// TIA Portal V19 export
FUNCTION_BLOCK "LAxisCtrlApcFr_Axis"   // FB19501, LAD
{ S7_Optimized_Access := 'TRUE' }
AUTHOR : APCFR
VERSION : 2.0
// V2.0.1
// stored: AutoNumber false, IsIECCheckEnabled true, MemoryReserve 100, SetENOAutomatically true
   VAR_INPUT
      enable : Bool := FALSE;
      stateSafetyActive : Bool := TRUE;   // STO or SOS active. Set FALSE if not used
      stateS120InfeedInOperation : Bool := FALSE;   // S120 infeed in operation input. Set TRUE if no infeed (AC/AC axis : CU310 or S210 or V90)
      enableAxis : Bool := FALSE;   // TRUE: Set axis enable; FALSE: Remove axis enable
      resetAxis : Bool := FALSE;   // Rising edge: Acknowledgement of technology alarms or restart of the axis (depending on configuration)
      openBrake : Bool := FALSE;
      jogForward : Bool := FALSE;   // Rising edge: Move an axis in jog mode (forward); Falling edge: Stop jogging
      jogBackward : Bool := FALSE;   // Rising edge: Move an axis in jog mode (backward); Falling edge: Stop jogging
      moveVelocity : Bool := FALSE;   // Rising edge: Move an axis at constant velocity/speed
      stop : Bool := FALSE;   // Rising edge: Brake an axis until it comes to a standstill
      eStop : Bool := FALSE;   // Emergency Stop with MC_Stop instruction
      torqueLimiting : Bool := FALSE;   // TRUE: Enable force/torque limiting
      homing : Bool := FALSE;   // Rising edge: Home axis
      homingToFixedStop : Bool := FALSE;
      homingOnSensor : Bool := FALSE;
      posRelative : Bool := FALSE;   // Rising edge: Move an axis relative to its position when execution of the job began
      posAbsolute : Bool := FALSE;   // Rising edge: Move an axis to an absolute position
      posSuperimposed : Bool := FALSE;   // Rising edge: Start a superimposed positioning
      haltSuperimposed : Bool := FALSE;
      gearInRelative : Bool := FALSE;
      gearInAbsolute : Bool := FALSE;
      gearInVelocity : Bool := FALSE;
      gearOutCamOut : Bool := FALSE;   // Rising edge: End a gearing/camming operation
      camIn : Bool := FALSE;
      camInStandStill : Bool := FALSE;
      camInChangeOnTheFly : Bool := FALSE;
      phasing : Bool := FALSE;
      offset : Bool := FALSE;   // Rising edge: Start an offset operation
      actDesactLimitSwitches : Bool := FALSE;
      changeModulo : Bool := FALSE;
      startEndLessMode : Bool := FALSE;
      simulationOnOff : Bool := FALSE;   // Rising edge starts action once
      resetMaxValues : Bool := FALSE;   // Reset max torque and max followingerror
      override : LReal := 100.0;   // Velocity override : 0 to 200%
      axis : DB_ANY;   // Reference to axis to be controlled
      master : DB_ANY;
      cam1 : DB_ANY;
      cam2 : DB_ANY;
      dataAxisConfig : "LAxisCtrlApcFr_typeAxisConfig";   // Structure for parameters
   END_VAR
   VAR_OUTPUT
      valid { ExternalWritable := 'False'} : Bool := FALSE;   // TRUE: Valid set of output values available at the FB
      busy { ExternalWritable := 'False'} : Bool := FALSE;
      error { ExternalWritable := 'False'} : Bool := FALSE;   // TRUE: An error occurred while processing the FB
      status { ExternalWritable := 'False'} : String := 'STATUS_NO_CALL';   // Current status of FB
      errorMC { ExternalWritable := 'False'} : String;
      errorID { ExternalWritable := 'False'} : String;
      driveReadyForOperation { ExternalWritable := 'False'} : Bool := FALSE;
      axisEnabled { ExternalWritable := 'False'} : Bool := FALSE;   // TRUE: The technology object is enabled. Motion commands can be executed
      axisHomed { ExternalWritable := 'False'} : Bool := FALSE;
      axisInPosition { ExternalWritable := 'False'} : Bool := FALSE;
      axisInStandstill { ExternalWritable := 'False'} : Bool := FALSE;
      axisInVelocity { ExternalWritable := 'False'} : Bool := FALSE;   // TRUE: The setpoint velocity/speed was reached and will be maintained
      axisInLimitation { ExternalWritable := 'False'} : Bool := FALSE;   // TRUE: The drive is operating at the force/torque limit
      axisInClamping { ExternalWritable := 'False'} : Bool := FALSE;   // TRUE: The drive is kept at the fixed stop (clamping), the axis position is within the positioning tolerance
      axisInSimulation : Bool := FALSE;
      axisCamInSelected { ExternalWritable := 'False'} : Bool := FALSE;
      axisInSynchronizing { ExternalWritable := 'False'} : Bool := FALSE;
      axisInSync { ExternalWritable := 'False'} : Bool := FALSE;
      camInStandStillDone { ExternalWritable := 'False'} : Bool := FALSE;
      camInStandStillBusy { ExternalWritable := 'False'} : Bool := FALSE;
      camInChangeOnTheFlyDone { ExternalWritable := 'False'} : Bool := FALSE;
      camInChangeOnTheFlylBusy { ExternalWritable := 'False'} : Bool := FALSE;
      eStopDone { ExternalWritable := 'False'} : Bool := FALSE;
      eStopBusy { ExternalWritable := 'False'} : Bool := FALSE;
      homingToFixedStopDone { ExternalWritable := 'False'} : Bool := FALSE;
      homingToFixedStopBusy { ExternalWritable := 'False'} : Bool := FALSE;
      homingOnSensorDone { ExternalWritable := 'False'} : Bool := FALSE;
      homingOnSensorBusy { ExternalWritable := 'False'} : Bool := FALSE;
      actDesactLimitSwitchesDone { ExternalWritable := 'False'} : Bool := FALSE;
      actDesactLimitSwitchesBusy { ExternalWritable := 'False'} : Bool := FALSE;
      changeModuloDone { ExternalWritable := 'False'} : Bool := FALSE;
      changeModuloBusy { ExternalWritable := 'False'} : Bool := FALSE;
      endLessModeDone { ExternalWritable := 'False'} : Bool := FALSE;
      endLessModeBusy { ExternalWritable := 'False'} : Bool := FALSE;
      simulationOnDone { ExternalWritable := 'False'} : Bool := FALSE;
      simulationOnBusy { ExternalWritable := 'False'} : Bool := FALSE;
      actualPosition { ExternalWritable := 'False'} : LReal;
      actualVelocity { ExternalWritable := 'False'} : LReal;
      actualSpeed { ExternalWritable := 'False'} : LReal;
      actualAcceleration { ExternalWritable := 'False'} : LReal;
      actualTorque { ExternalWritable := 'False'} : LReal;
      actualTorqueMax { ExternalWritable := 'False'} : LReal;
      actualFollowingError { ExternalWritable := 'False'} : LReal;
      actualFollowingErrorMax { ExternalWritable := 'False'} : LReal;
      camSelected { ExternalWritable := 'False'} : UInt;
      camUsed { ExternalWritable := 'False'} : UInt;
      HistoricBuffer { ExternalWritable := 'False'} : "LAxisCtrlApcFr_typeHistoricBufferCmd";
      outputsLAxisCtrl_Axis { ExternalWritable := 'False'} : Struct
         valid : Bool := FALSE;   // TRUE: Valid set of output values available at the FB
         busy : Bool := FALSE;   // TRUE: FB is working and new output values can be expected
         error : Bool := FALSE;   // TRUE: An error occurred while processing the FB
         status : Word;   // Current status of FB (16#0000 - 16#7FFF: Status of the FB, 16#8000 - 16#FFFF: Error identification)
         statusText : String := STRING#'STATUS_NO_CALL';   // Text of current status of FB
         subfunctionStatus : Word;   // Status of internally called subfunctions (ErrorID of Motion Control instructions)
         axisEnabled : Bool := FALSE;   // TRUE: The technology object is enabled. Motion commands can be executed
         resetActive : Bool := FALSE;   // TRUE: Reset/Restart of the axis is active
         commandBusy : Bool := FALSE;   // TRUE: The selected basic motion command is being executed
         commandDone : Bool := FALSE;   // TRUE: The selected basic motion command has completed without error
         commandAborted : Bool := FALSE;   // TRUE: The selected basic motion command has been aborted
         inVelocity : Bool := FALSE;   // TRUE: The setpoint velocity/speed was reached and will be maintained
         inLimitation : Bool := FALSE;   // TRUE: The drive is operating at the force/torque limit
         homingCommandBusy : Bool := FALSE;   // TRUE: Homing command is being executed
         homingCommandDone : Bool := FALSE;   // TRUE: Homing command has completed without error
         homingCommandAborted : Bool := FALSE;   // TRUE: Homing command has been aborted
         superimposedBusy : Bool := FALSE;   // TRUE: The selected superimposed motion command is being executed
         superimposedDone : Bool := FALSE;   // TRUE: The selected superimposed motion command has completed without error
         superimposedAborted : Bool := FALSE;   // TRUE: The selected superimposed motion command has been aborted
         superimposedStart : Bool := FALSE;   // TRUE: The selected superimposed motion is active
         inClamping : Bool := FALSE;   // TRUE: The drive is kept at the fixed stop (clamping), the axis position is within the positioning tolerance
         startSync : Bool := FALSE;   // TRUE: The axis is synchronizing to the leading axis / desynchronizing from the leading axis (Note: signal is only valid for the currently selected synchronous functionality, see outputs 'gearInRelativeSelected', 'gearInAbsoluteSelected', 'gearInVelocitySelected', 'gearOutCamOutSelected' or 'camInSelected')
         inSync : Bool := FALSE;   // TRUE: The axis is synchronized to the leading axis (Note: signal is only valid for the currently selected synchronous functionality, see outputs 'gearInRelativeSelected', 'gearInAbsoluteSelected', 'gearInVelocitySelected' or 'camInSelected')
         endOfProfile : Bool := FALSE;   // TRUE: The end of the cam has been reached. The output is displayed for at least one call when the cam is used cyclically
         inSimulation : Bool := FALSE;   // TRUE: Synchronous operation is being simulated
         jogSelected : Bool := FALSE;   // TRUE: Jogging is active
         moveVelocitySelected : Bool := FALSE;   // TRUE: Moving with constant velocity/speed is active
         stopSelected : Bool := FALSE;   // TRUE: Stopping is active
         fastStopSelected : Bool := FALSE;   // TRUE: Stopping is active (with fastStop dynamics)
         torqueLimitingSelected : Bool := FALSE;   // TRUE: Force/Torque limiting is active
         homingSelected : Bool := FALSE;   // TRUE: Homing is active
         posRelativeSelected : Bool := FALSE;   // TRUE: Relative positioning is active
         posAbsoluteSelected : Bool := FALSE;   // TRUE: Absolute positioning is active
         posSuperimposedSelected : Bool := FALSE;   // TRUE: Superimposed positioning is active (See also outputs: superimposedBusy, superimposedDone, superimposedAborted)
         haltSuperimposedSelected : Bool := FALSE;   // TRUE: Superimposed halting is active (See also outputs: superimposedBusy, superimposedDone, superimposedAborted)
         gearInRelativeSelected : Bool := FALSE;   // TRUE: Relative gearing is active (See also outputs: commandBusy, commandDone, commandAborted, inSync)
         gearInAbsoluteSelected : Bool := FALSE;   // TRUE: Absolute gearing is active (See also outputs: commandBusy, commandDone, commandAborted, startSync, inSync)
         gearInVelocitySelected : Bool := FALSE;   // TRUE: Velocity gearing is active (See also outputs: commandBusy, commandDone, commandAborted, startSync, inSync)
         gearOutCamOutSelected : Bool := FALSE;   // TRUE: End a gearing/camming operation is active (See also outputs: commandBusy, commandDone, commandAborted, startSync)
         camInSelected : Bool := FALSE;   // TRUE: Camming is active (See also outputs: commandBusy, commandDone, commandAborted, startSync, inSync)
         phasingSelected : Bool := FALSE;   // TRUE: Phasing is active (See also outputs: superimposedBusy, superimposedDone, superimposedAborted, superimposedStart)
         offsetSelected : Bool := FALSE;   // TRUE: Offset is active (See also outputs: superimposedBusy, superimposedDone, superimposedAborted, superimposedStart)
         diagnostics : "LAxisCtrl_typeDiagnostics";   // Diagnostics structure
      END_STRUCT;
      outputsStatusWordTO { ExternalWritable := 'False'} : Struct
         enable : Bool;   // TRUE: The technology object has been enabled
         error : Bool;   // TRUE: An error is present
         restartActive : Bool;   // TRUE: A restart is active. The technology object is being reinitialized
         onlineStartValuesChanged : Bool;   // TRUE: The restart tags have been changed. For the changes to be applied, the technology object must be reinitialized
         controlPanelActive : Bool;   // TRUE: The axis control panel is active
         homingDone : Bool;   // TRUE: The technology object is homed
         done : Bool;   // TRUE: No motion job is in progress and the axis control panel is deactivated
         standstill : Bool;   // TRUE: The axis is at a standstill
         positioningCommand : Bool;   // TRUE: A positioning command is active ("MC_MoveRelative", "MC_MoveAbsolute")
         jogCommand : Bool;   // TRUE: An "MC_MoveJog" job is running
         velocityCommand : Bool;   // TRUE: An "MC_MoveVelocity" job is running
         homingCommand : Bool;   // TRUE: An "MC_Home" job is being processed
         constantVelocity : Bool;   // TRUE: The velocity setpoint is reached. A constant velocity setpoint is output
         accelerating : Bool;   // TRUE: An acceleration operation is active
         decelerating : Bool;   // TRUE: A deceleration operation is active
         swLimitMinActive : Bool;   // TRUE: A negative software limit switch has been approached or exceeded
         swLimitMaxActive : Bool;   // TRUE: A positive software limit switch has been approached or exceeded
         hwLimitMinActive : Bool;   // TRUE: A negative hardware limit switch has been approached or exceeded
         hwLimitMaxActive : Bool;   // TRUE: A positive hardware limit switch has been approached or exceeded
         synchronizing : Bool;   // TRUE: The axis synchronizes to a leading value
         synchronous : Bool;   // TRUE: The axis moves synchronously to a leading value
         superimposedMotionCommand : Bool;   // TRUE: An "MC_MoveSuperimposed" job is running
         phasingCommand : Bool;   // TRUE: An "MC_PhasingAbsolute" or "MC_PhasingRelative" job for the leading value shift is active
         axisSimulation : Bool;   // TRUE: The technology object is in simulation
         torqueLimitingCommand : Bool;   // TRUE: An "MC_TorqueLimiting" job is running
         inLimitation : Bool;   // TRUE: The drive operates at least at the threshold value (default 90%) of the torque limit/force limitation
         nonPositionControlled : Bool;   // TRUE: The axis is not in position-controlled mode
         kinematicsMotionCommand : Bool;   // TRUE: The axis is used for a kinematics job
         inClamping : Bool;   // TRUE: The axis is clamped at a fixed stop
         motionInCommand : Bool;   // TRUE: An "MC_MotionIn" job is active
         stopCommand : Bool;   // TRUE: An "MC_Stop" job is running. The technology object is locked
         desynchronizingCommand : Bool;   // TRUE: An "MC_GearOut" job or "MC_CamOut" job is active. The following axis is desynchronized
         passingBacklash : Bool;   // TRUE: The backlash is traversed. <TO>.ActualPosition does not hereby change
         phasingCommandWaiting : Bool;   // TRUE: An "MC_PhasingAbsolute" or "MC_PhasingRelative" job for leading value shift is waiting
         offsetCommand : Bool;   // TRUE: An "MC_OffsetAbsolute" or "MC_OffsetRelative" job for following value offset is active
         offsetCommandWaiting : Bool;   // TRUE: An "MC_OffsetAbsolute" or "MC_OffsetRelative" job for following value offset is waiting
         motionInSuperimposedCommand : Bool;   // TRUE: An "MC_MotionInSuperimposed" job is running
         haltSuperimposedCommand : Bool;   // TRUE: An "MC_HaltSuperimposed" job is running
      END_STRUCT;
   END_VAR
   VAR
      statFirstCall { ExternalAccessible := 'False'; ExternalVisible := 'False'; ExternalWritable := 'False'} : Bool;   // TRUE: First call of FB
      statLastCall { ExternalAccessible := 'False'; ExternalVisible := 'False'; ExternalWritable := 'False'} : Bool;
      statEnableOld { ExternalAccessible := 'False'; ExternalVisible := 'False'; ExternalWritable := 'False'} : Bool;   // Old value of enable for edge detection
      statErrorLAxisCtrlStd { ExternalAccessible := 'False'; ExternalVisible := 'False'; ExternalWritable := 'False'} : Bool;
      statErrorActDesactLimitSwitches { ExternalAccessible := 'False'; ExternalVisible := 'False'; ExternalWritable := 'False'} : Bool;
      statErrorChangeModuloAxis { ExternalAccessible := 'False'; ExternalVisible := 'False'; ExternalWritable := 'False'} : Bool;
      statErrorHomingToFixedStop { ExternalAccessible := 'False'; ExternalVisible := 'False'; ExternalWritable := 'False'} : Bool;
      statErrorHomingOnSensor { ExternalAccessible := 'False'; ExternalVisible := 'False'; ExternalWritable := 'False'} : Bool;
      statErrorEndLessMode { ExternalAccessible := 'False'; ExternalVisible := 'False'; ExternalWritable := 'False'} : Bool;
      statErrorSimulationOnOff { ExternalAccessible := 'False'; ExternalVisible := 'False'; ExternalWritable := 'False'} : Bool;
      statErrorCamInStandStill { ExternalAccessible := 'False'; ExternalVisible := 'False'; ExternalWritable := 'False'} : Bool;
      statErrorCamSelection { ExternalAccessible := 'False'; ExternalVisible := 'False'; ExternalWritable := 'False'} : Bool;
      statErrorCamStandStillSelection { ExternalAccessible := 'False'; ExternalVisible := 'False'; ExternalWritable := 'False'} : Bool;
      statErrorInterpolateCam { ExternalAccessible := 'False'; ExternalVisible := 'False'; ExternalWritable := 'False'} : Bool;
      statErrorCamIChangeOnTheFly { ExternalAccessible := 'False'; ExternalVisible := 'False'; ExternalWritable := 'False'} : Bool;
      statErrorGearInPos { ExternalAccessible := 'False'; ExternalVisible := 'False'; ExternalWritable := 'False'} : Bool;
      statErrorEStop { ExternalAccessible := 'False'; ExternalVisible := 'False'; ExternalWritable := 'False'} : Bool;
      statFirstError { ExternalAccessible := 'False'; ExternalVisible := 'False'; ExternalWritable := 'False'} : Bool;
      returnValueRD_LOC_T { ExternalAccessible := 'False'; ExternalVisible := 'False'; ExternalWritable := 'False'} : Int;
      statEnableAxisOld { ExternalAccessible := 'False'; ExternalVisible := 'False'; ExternalWritable := 'False'} : Bool := FALSE;   // TRUE: Set axis enable; FALSE: Remove axis enable
      statHomingOld { ExternalAccessible := 'False'; ExternalVisible := 'False'; ExternalWritable := 'False'} : Bool := FALSE;   // Rising edge: Home axis
      statIndex { ExternalAccessible := 'False'; ExternalVisible := 'False'; ExternalWritable := 'False'} : Int;
      statHistoricBuffer { ExternalAccessible := 'False'; ExternalVisible := 'False'; ExternalWritable := 'False'} : "LAxisCtrlApcFr_typeHistoricBufferCmd";
      statAxisName { ExternalAccessible := 'False'; ExternalVisible := 'False'; ExternalWritable := 'False'} : WString;
      statDiagnostic { ExternalAccessible := 'False'; ExternalVisible := 'False'; ExternalWritable := 'False'} : Struct
         status : Word;
         errorMC : Word;
         errorID : Word;
      END_STRUCT;
      statReset { ExternalAccessible := 'False'; ExternalVisible := 'False'; ExternalWritable := 'False'} : Bool;
      statOpenBrake { ExternalAccessible := 'False'; ExternalVisible := 'False'; ExternalWritable := 'False'} : Bool;
      statStop { ExternalAccessible := 'False'; ExternalVisible := 'False'; ExternalWritable := 'False'} : Bool;
      statFastStop { ExternalAccessible := 'False'; ExternalVisible := 'False'; ExternalWritable := 'False'} : Bool;
      statEStop { ExternalAccessible := 'False'; ExternalVisible := 'False'; ExternalWritable := 'False'} : Bool;
      statTorqueLimiting { ExternalAccessible := 'False'; ExternalVisible := 'False'; ExternalWritable := 'False'} : Bool;
      statHoming { ExternalAccessible := 'False'; ExternalVisible := 'False'; ExternalWritable := 'False'} : Bool;
      statJogForward { ExternalAccessible := 'False'; ExternalVisible := 'False'; ExternalWritable := 'False'} : Bool;
      statJogBackward { ExternalAccessible := 'False'; ExternalVisible := 'False'; ExternalWritable := 'False'} : Bool;
      statMoveVelocity { ExternalAccessible := 'False'; ExternalVisible := 'False'; ExternalWritable := 'False'} : Bool;
      statPosRelative { ExternalAccessible := 'False'; ExternalVisible := 'False'; ExternalWritable := 'False'} : Bool;
      statPosAbsolute { ExternalAccessible := 'False'; ExternalVisible := 'False'; ExternalWritable := 'False'} : Bool;
      statSuperimposed { ExternalAccessible := 'False'; ExternalVisible := 'False'; ExternalWritable := 'False'} : Bool;
      statHaltSuperimposed { ExternalAccessible := 'False'; ExternalVisible := 'False'; ExternalWritable := 'False'} : Bool;
      statGearInVelocity { ExternalAccessible := 'False'; ExternalVisible := 'False'; ExternalWritable := 'False'} : Bool;
      statGearInRelative { ExternalAccessible := 'False'; ExternalVisible := 'False'; ExternalWritable := 'False'} : Bool;
      statGearInAbsolute { ExternalAccessible := 'False'; ExternalVisible := 'False'; ExternalWritable := 'False'} : Bool;
      statCamIn { ExternalAccessible := 'False'; ExternalVisible := 'False'; ExternalWritable := 'False'} : Bool;
      statCamInStandStill { ExternalAccessible := 'False'; ExternalVisible := 'False'; ExternalWritable := 'False'} : Bool;
      statCamInChangeOnTheFly { ExternalAccessible := 'False'; ExternalVisible := 'False'; ExternalWritable := 'False'} : Bool;
      statGearOutCamOut { ExternalAccessible := 'False'; ExternalVisible := 'False'; ExternalWritable := 'False'} : Bool;
      statPhasing { ExternalAccessible := 'False'; ExternalVisible := 'False'; ExternalWritable := 'False'} : Bool;
      statOffset { ExternalAccessible := 'False'; ExternalVisible := 'False'; ExternalWritable := 'False'} : Bool;
      statCam { ExternalAccessible := 'False'; ExternalVisible := 'False'; ExternalWritable := 'False'} : DB_ANY;
      statCamStandStill { ExternalAccessible := 'False'; ExternalVisible := 'False'; ExternalWritable := 'False'} : DB_ANY;
      statCamStanStillSelected { ExternalAccessible := 'False'; ExternalVisible := 'False'; ExternalWritable := 'False'} : UInt;
      statActDesactLimitSwitches { ExternalAccessible := 'False'; ExternalVisible := 'False'; ExternalWritable := 'False'} : Bool;
      statChangeModulo { ExternalAccessible := 'False'; ExternalVisible := 'False'; ExternalWritable := 'False'} : Bool;
      statHomingToFixedStop { ExternalAccessible := 'False'; ExternalVisible := 'False'; ExternalWritable := 'False'} : Bool;
      statHomingOnSensor { ExternalAccessible := 'False'; ExternalVisible := 'False'; ExternalWritable := 'False'} : Bool;
      statStartEndLessMode { ExternalAccessible := 'False'; ExternalVisible := 'False'; ExternalWritable := 'False'} : Bool;
      statSimulationOnOff { ExternalAccessible := 'False'; ExternalVisible := 'False'; ExternalWritable := 'False'} : Bool;
      statDataAxisConfigLAxisCtrl { ExternalAccessible := 'False'; ExternalVisible := 'False'; ExternalWritable := 'False'} : "LAxisCtrl_typeAxisConfig";
      statOffsetChangeOnTheFly { ExternalAccessible := 'False'; ExternalVisible := 'False'; ExternalWritable := 'False'} : LReal;
      statAxisCommandStatusDWord : DWord;
      instLAxisCtrl_Axis { ExternalAccessible := 'False'; ExternalVisible := 'False'; ExternalWritable := 'False'} : "LAxisCtrl_Axis";
      instLAxisCtrl_AxisStatusWord { ExternalAccessible := 'False'; ExternalVisible := 'False'; ExternalWritable := 'False'} : "LAxisCtrl_AxisStatusWord";
      instLAxisCtrlApcFr_CamInStandStill { ExternalAccessible := 'False'; ExternalVisible := 'False'; ExternalWritable := 'False'} : "LAxisCtrlApcFr_CamInStandStill";
      instLAxisCtrlApcFr_GetCamStatusWord { ExternalAccessible := 'False'; ExternalVisible := 'False'; ExternalWritable := 'False'} : "LAxisCtrlApcFr_UnpubGetCamStatusWord";
      InstLAxisCtrlApcFr_McGearInPos_Axis { ExternalAccessible := 'False'; ExternalVisible := 'False'; ExternalWritable := 'False'} : "LAxisCtrlApcFr_McGearInPos_Axis";
      instLAxisCtrlApcFr_HystoricBuffer { ExternalAccessible := 'False'; ExternalVisible := 'False'; ExternalWritable := 'False'} : "LAxisCtrlApcFr_HystoricBuffer";
      instLAxisCtrlApcFr_UnpubAxis_eSTOP { ExternalAccessible := 'False'; ExternalVisible := 'False'; ExternalWritable := 'False'} : "LAxisCtrlApcFr_UnpubAxis_eSTOP";
      instLaxisCtrlApcFr_GetCommandAxisStatusDWord { ExternalAccessible := 'False'; ExternalVisible := 'False'; ExternalWritable := 'False'} : "LAxisCtrlApcFr_GetCommandAxisStatusDWord";
      instLaxisCtrlApcFr_UnpubMC_Interpolate { ExternalAccessible := 'False'; ExternalVisible := 'False'; ExternalWritable := 'False'} : "LAxisCtrlApcFr_UnpubMC_Interpolate";
      instLAxisCtrlApcFr_ActDeactLimitSwitches { ExternalAccessible := 'False'; ExternalVisible := 'False'; ExternalWritable := 'False'} : "LAxisCtrlApcFr_ActDeactLimitSwitches";
      instLAxisCtrlApcFr_ChangeModulo { ExternalAccessible := 'False'; ExternalVisible := 'False'; ExternalWritable := 'False'} : "LAxisCtrlApcFr_ChangeModulo";
      instLAxisCtrlApcFr_HomingToFixedStop { ExternalAccessible := 'False'; ExternalVisible := 'False'; ExternalWritable := 'False'} : "LAxisCtrlApcFr_HomingToFixedStop";
      instAxisCtrlAapcFr_HomingOnSensor { ExternalAccessible := 'False'; ExternalVisible := 'False'; ExternalWritable := 'False'} : "LAxisCtrlApcFr_HomingOnSensor";
      instLAxisCtrlApcFr_EndLessMode { ExternalAccessible := 'False'; ExternalVisible := 'False'; ExternalWritable := 'False'} : "LAxisCtrlApcFr_EndLessMode";
      instLAxisCtrlApcFR_SimulationOnOff { ExternalAccessible := 'False'; ExternalVisible := 'False'; ExternalWritable := 'False'} : "LAxisCtrlApcFr_SimulationOnOff";
      instLaxisCtrlApcFr_CamInChangeOnTheFly { ExternalAccessible := 'False'; ExternalVisible := 'False'; ExternalWritable := 'False'} : "LAxisCtrlApcFr_CamInChangeOnTheFly";
      statAxis { ExternalAccessible := 'False'; ExternalVisible := 'False'; ExternalWritable := 'False'} : DB_ANY;
      statMaster { ExternalAccessible := 'False'; ExternalVisible := 'False'; ExternalWritable := 'False'} : DB_ANY;
      statCommunicationOK { ExternalAccessible := 'False'; ExternalVisible := 'False'; ExternalWritable := 'False'} : Bool;
   END_VAR
   VAR_TEMP
      tempVoidBool : Bool;   // Temp value for operative sensor
      tempAbsActualTorque : LReal;
      tempAbsActualTorqueMax : LReal;
      tempRefCamBase2 : REF_TO TO_CamBase;   // Temporary reference of the technology object type TO_CamBase
      tempRefCamBase1 : REF_TO TO_CamBase;   // Temporary reference of the technology object type TO_CamBase
      tempRefAxis : REF_TO TO_Axis;   // Temporary reference of the technology object type TO_Axis
      tempRefSpeedAxis : REF_TO TO_SpeedAxis;   // Temporary reference of the technology object type TO_SpeedAxis
      tempRefPosAxis : REF_TO TO_PositioningAxis;   // Temporary reference of the technology object type TO_PositioningAxis
      tempRefSyncAxis : REF_TO TO_SynchronousAxis;   // Temporary reference of the technology object type TO_PositioningAxis
      tempReturnValue : Int;
      tempDateAndTime : Date_And_Time;
      tempDateOfDay : Time_Of_Day;
   END_VAR
   VAR_TEMP   // added for the SCL form of the ladder/FBD networks
      _w1 : Bool;
   END_VAR
BEGIN

REGION Network 1 (SCL): (** COMMENTS **)
   //===================================================================================================
   // SIEMENS SAS    RC-FR DI FA APC
   //---------------------------------------------------------------------------------------------------
   // Restrictions:  TIA V16 or more in function of library version
   // Requirements:  S7-1500 + LAxisCtrl library
   //---------------------------------------------------------------------------------------------------
   // Description:   This function block offers basic functionalities for TO SynchronousAxis
   //                based on LAxisCtrl_SyncAxisCamming with additionnals functionalities
   //---------------------------------------------------------------------------------------------------
   // Change log table:
   // Version  Date        TIA   Expert  Changes applied
   // 01.xx    2020.07.24  V16   SDA     see LaxisCtrlApcFr_aVersion 
   // 02.xx    2021.10.18  V17   SDA     see LaxisCtrlApcFr_aVersion 
   // 03.xx    2024.09.12  V19   SDA     see LaxisCtrlApcFr_aVersion
   //---------------------------------------------------------------------------------------------------
   // Compatibility to TIA version require the use of latest version for PLC fimware and Motion Control 
   // e.g: Firmware 3.1 and Motion Control V7.0 for TIA V19
   //===================================================================================================
END_REGION

REGION Network 2 (SCL): (** INIT **)
   //----------------------------------------------------------------------------------------------
   #statFirstCall := #enable AND NOT #statEnableOld;
   #statLastCall := NOT #enable AND #statEnableOld;
   #statEnableOld := #enable;

   #tempRefAxis ?= #master;
   #tempRefSyncAxis ?= #axis;
   #tempRefCamBase1 ?= #cam1;
   #tempRefCamBase2 ?= #cam2;

   #statAxis := #axis;
   #statMaster := #master;

   IF #statFirstCall THEN
       REGION InitFirstCall
           // #statAxisName := GetSymbolPath(variable := #axis, size := 36);
           // "LaxisCtrlApcFr_GetPosSyncAxisGeneralValues"(axis := #axis,
           // axisGeneral := #dataAxisConfig.axisGeneral);
           // Diagnostic in string
           #status := 'STATUS_FIRST_CALL';
           #error := FALSE;
           #errorMC := 'No errorMC';
           #errorID := 'No errorID';
           // Diagnostic in word
           #statDiagnostic.status := "STATUS_FIRST_CALL";
           #statDiagnostic.errorMC := "STATUS_FINISHED_NOERROR";
           #statDiagnostic.errorID := "STATUS_FINISHED_NOERROR";

           #statFirstError := FALSE;

           #statAxis := #axis;
           #statMaster := #master;
           RETURN;
       END_REGION

   ELSIF #statLastCall THEN
       REGION InitLastCall
           // Reset outputs
           REGION Reset outputs 
               #error := FALSE;
               #status := 'STATUS_LAST_CALL';
               #errorMC := 'No ErrorMC';
               #statDiagnostic.status := "STATUS_FINISHED_NOERROR";
               #statDiagnostic.errorMC := "STATUS_FINISHED_NOERROR";
               #driveReadyForOperation := FALSE;
               #axisInPosition := FALSE;
               #axisInStandstill := FALSE;
               #axisInVelocity := FALSE;
               #axisInLimitation := FALSE;
               #axisInClamping := FALSE;
               #axisCamInSelected := FALSE;
               #axisInSynchronizing := FALSE;
               #camInStandStillDone := FALSE;
               #camInStandStillBusy := FALSE;
               #camInChangeOnTheFlyDone := FALSE;
               #camInChangeOnTheFlylBusy := FALSE;
               #axisInSync := FALSE;
               #eStopDone := FALSE;
               #eStopBusy := FALSE;
               #homingToFixedStopDone := FALSE;
               #homingToFixedStopBusy := FALSE;
               #homingOnSensorDone := FALSE;
               #homingOnSensorBusy := FALSE;
               #actDesactLimitSwitchesDone := FALSE;
               #actDesactLimitSwitchesBusy := FALSE;
               #changeModuloDone := FALSE;
               #changeModuloBusy := FALSE;
               #endLessModeDone := FALSE;
               #endLessModeBusy := FALSE;
               #simulationOnDone := FALSE;
               #simulationOnBusy := FALSE;
               #actualPosition := 0.0;
               #actualVelocity := 0.0;
               #actualSpeed := 0.0;
               #actualAcceleration := 0.0;
               #actualTorque := 0.0;
               #actualTorqueMax := 0.0;
               #actualFollowingError := 0.0;
               #actualFollowingErrorMax := 0.0;
           END_REGION

           // Reset internal variables
           REGION Reset internal variables
               #statFirstCall := FALSE;
               #statLastCall := FALSE;
               #statEnableOld := FALSE;
               #statErrorLAxisCtrlStd := FALSE;
               #statErrorActDesactLimitSwitches := FALSE;
               #statErrorChangeModuloAxis := FALSE;
               #statErrorHomingToFixedStop := FALSE;
               #statErrorHomingOnSensor := FALSE;
               #statErrorEndLessMode := FALSE;
               #statErrorEStop := FALSE;
               #statFirstError := FALSE;
               #statEnableAxisOld := FALSE;
               #statHomingOld := FALSE;
               #statIndex := 0;
               #statReset := FALSE;
               #statOpenBrake := FALSE;
               #statStop := FALSE;
               #statFastStop := FALSE;
               #statEStop := FALSE;
               #statTorqueLimiting := FALSE;
               #statHoming := FALSE;
               #statJogForward := FALSE;
               #statJogBackward := FALSE;
               #statMoveVelocity := FALSE;
               #statPosRelative := FALSE;
               #statPosAbsolute := FALSE;
               #statSuperimposed := FALSE;
               #statHaltSuperimposed := FALSE;
               #statGearInRelative := FALSE;
               // cpu-t functions
               #statGearInVelocity := FALSE;
               #statGearInAbsolute := FALSE;
               #statGearInAbsolute := FALSE;
               #statCamInStandStill := FALSE;
               #statCamInChangeOnTheFly := FALSE;
               #statGearOutCamOut := FALSE;
               #statPhasing := FALSE;
               #statOffset := FALSE;
               // additionnal functions
               #statActDesactLimitSwitches := FALSE;
               #statChangeModulo := FALSE;
               #statHomingToFixedStop := FALSE;
               #statHomingOnSensor := FALSE;
               #statStartEndLessMode := FALSE;
               #statSimulationOnOff := FALSE;
           END_REGION

           //RETURN;
       END_REGION

   ELSIF NOT #enable AND NOT #instLAxisCtrl_Axis.busy THEN
       REGION NotEnable

           #error := FALSE;
           // Diagnostic in string
           #status := 'STATUS_NO_CALL';
           #errorMC := 'No errorMC';
           #errorID := 'No errorID';
           // Diagnostic in word
           #statDiagnostic.status := "STATUS_NO_CALL";
           #statDiagnostic.errorMC := "STATUS_FINISHED_NOERROR";
           #statDiagnostic.errorID := "STATUS_FINISHED_NOERROR";
           #statFirstError := FALSE;

           RETURN;
       END_REGION
   END_IF;

   IF NOT #error THEN
       #status := 'STATUS_CALL_FB';
       #errorMC := 'No errorMC';
       #statDiagnostic.status := "STATUS_FINISHED_NOERROR";
       #statDiagnostic.errorMC := "STATUS_FINISHED_NOERROR";
   END_IF;
   //----------------------------------------------------------------------------------------------
END_REGION

REGION Network 3 (SCL): (** COMMAND **)
   IF #enable AND NOT #error THEN
       #statReset := #resetAxis;
       #statOpenBrake := #openBrake;
       #statStop := #stop;
       //#statFastStop := #fastStop;
       #statTorqueLimiting := #torqueLimiting;
       #statHoming := #homing;
       #statJogForward := #jogForward;
       #statJogBackward := #jogBackward;
       #statMoveVelocity := #moveVelocity;
       #statPosRelative := #posRelative;
       #statPosAbsolute := #posAbsolute;
       #statSuperimposed := #posSuperimposed;
       #statHaltSuperimposed := #haltSuperimposed;
       #statGearInRelative := #gearInRelative;
       #statCamIn := #camIn;
       #statGearOutCamOut := #gearOutCamOut;
       #statPhasing := #phasing;
       #statOffset := #offset;

       #statGearInAbsolute := #gearInAbsolute;
       #statGearInVelocity := #gearInVelocity;
       #statCamInStandStill := #camInStandStill;
       #statCamInChangeOnTheFly := #camInChangeOnTheFly;
       #statEStop := #eStop;
       #statActDesactLimitSwitches := #actDesactLimitSwitches;
       #statChangeModulo := #changeModulo;
       #statHomingToFixedStop := #homingToFixedStop;
       #statHomingOnSensor := #homingOnSensor;
       #statStartEndLessMode := #startEndLessMode;
       #statSimulationOnOff := #simulationOnOff;

   ELSIF #error THEN
       #statReset := #resetAxis;
       #statOpenBrake := #openBrake;
       #statStop := #stop;
       //#statFastStop := #fastStop;
       #statTorqueLimiting := FALSE;
       #statHoming := FALSE;
       #statJogForward := FALSE;
       #statJogBackward := FALSE;
       #statMoveVelocity := FALSE;
       #statPosRelative := FALSE;
       #statPosAbsolute := FALSE;
       #statSuperimposed := FALSE;
       #statHaltSuperimposed := FALSE;

       #statGearInRelative := FALSE;
       #statCamIn := FALSE;
       #statGearOutCamOut := FALSE;
       #statPhasing := FALSE;
       #statOffset := FALSE;

       #statGearInAbsolute := FALSE;
       #statGearInVelocity := FALSE;
       #statCamInStandStill := FALSE;
       #statCamInChangeOnTheFly := FALSE;
       #statEStop := #eStop;
       #statActDesactLimitSwitches := FALSE;
       #statChangeModulo := FALSE;
       #statHomingToFixedStop := FALSE;
       #statHomingOnSensor := FALSE;
       #statStartEndLessMode := FALSE;
       #statSimulationOnOff := FALSE;

    ELSE
        #statReset := FALSE;
        #statOpenBrake := FALSE;
        #statStop := FALSE;
        #statFastStop := FALSE;
        #statEStop := false;
        #statTorqueLimiting := FALSE;
        #statHoming := FALSE;
        #statJogForward := FALSE;
        #statJogBackward := FALSE;
        #statMoveVelocity := FALSE;
        #statPosRelative := FALSE;
        #statPosAbsolute := FALSE;
        #statSuperimposed := FALSE;
        #statHaltSuperimposed := FALSE;

        #statGearInRelative := FALSE;
        #statCamIn := FALSE;
        #statGearOutCamOut := FALSE;
        #statPhasing := FALSE;
        #statOffset := FALSE;

        #statGearInAbsolute := FALSE;
        #statGearInVelocity := FALSE;
        #statCamInStandStill := FALSE;
        #statCamInChangeOnTheFly := FALSE;
        #statEStop := FALSE;
        #statActDesactLimitSwitches := FALSE;
        #statChangeModulo := FALSE;
        #statHomingToFixedStop := FALSE;
        #statHomingOnSensor := FALSE;
        #statStartEndLessMode := FALSE;
        #statSimulationOnOff := FALSE;

   END_IF;
END_REGION

REGION Network 4: (** INTERPOLATE CAM **) / (** HISTORIC BUFFER **)
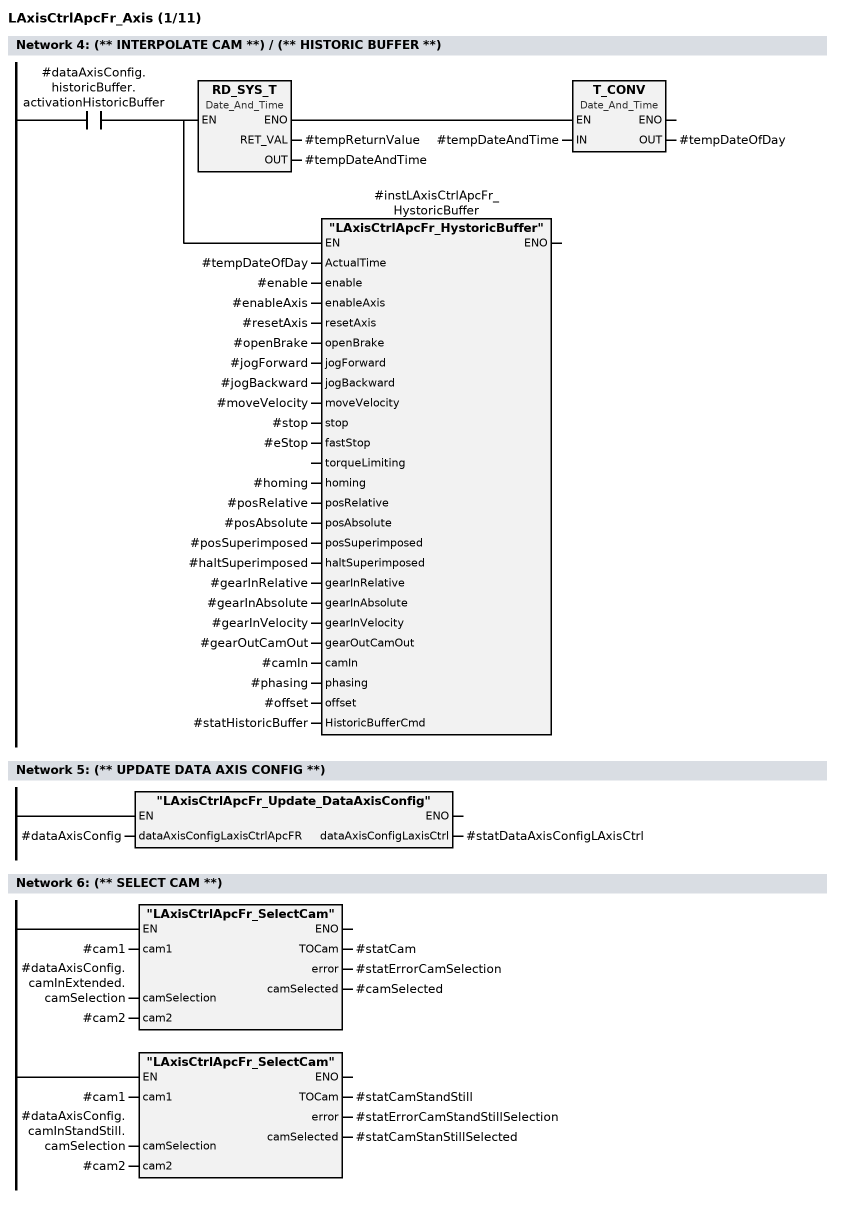
   RUNG wire#powerrail
      Contact( #dataAxisConfig.historicBuffer.activationHistoricBuffer )
      wire#w1
      { S7_Templates := "date_type := Date_And_Time" } RD_SYS_T(RET_VAL => #tempReturnValue, OUT => #tempDateAndTime)
      { S7_Templates := "[src_type := Date_And_Time, dest_type := Time_Of_Day]" } T_CONV(IN := #tempDateAndTime, OUT => #tempDateOfDay)
   END_RUNG
   RUNG wire#w1
      #instLAxisCtrlApcFr_HystoricBuffer(ActualTime := #tempDateOfDay, enable := #enable, enableAxis := #enableAxis, resetAxis := #resetAxis, openBrake := #openBrake, jogForward := #jogForward, jogBackward := #jogBackward, moveVelocity := #moveVelocity, stop := #stop, fastStop := #eStop, torqueLimiting :=, homing := #homing, posRelative := #posRelative, posAbsolute := #posAbsolute, posSuperimposed := #posSuperimposed, haltSuperimposed := #haltSuperimposed, gearInRelative := #gearInRelative, gearInAbsolute := #gearInAbsolute, gearInVelocity := #gearInVelocity, gearOutCamOut := #gearOutCamOut, camIn := #camIn, phasing := #phasing, offset := #offset, HistoricBufferCmd := #statHistoricBuffer)
   END_RUNG
   // the same network as SCL:
   #tempReturnValue := RD_SYS_T(EN := #dataAxisConfig.historicBuffer.activationHistoricBuffer,
                           OUT => #tempDateAndTime,
                           ENO => #_w1);
   IF #_w1 THEN T_CONV(IN := #tempDateAndTime, OUT => #tempDateOfDay); END_IF;
   IF #dataAxisConfig.historicBuffer.activationHistoricBuffer THEN
       #instLAxisCtrlApcFr_HystoricBuffer(ActualTime := #tempDateOfDay,   // "LAxisCtrlApcFr_HystoricBuffer"
                               enable := #enable,
                               enableAxis := #enableAxis,
                               resetAxis := #resetAxis,
                               openBrake := #openBrake,
                               jogForward := #jogForward,
                               jogBackward := #jogBackward,
                               moveVelocity := #moveVelocity,
                               stop := #stop,
                               fastStop := #eStop,
                               homing := #homing,
                               posRelative := #posRelative,
                               posAbsolute := #posAbsolute,
                               posSuperimposed := #posSuperimposed,
                               haltSuperimposed := #haltSuperimposed,
                               gearInRelative := #gearInRelative,
                               gearInAbsolute := #gearInAbsolute,
                               gearInVelocity := #gearInVelocity,
                               gearOutCamOut := #gearOutCamOut,
                               camIn := #camIn,
                               phasing := #phasing,
                               offset := #offset,
                               HistoricBufferCmd := #statHistoricBuffer);
   END_IF;
END_REGION

REGION Network 5: (** UPDATE DATA AXIS CONFIG **)
   RUNG wire#powerrail
      "LAxisCtrlApcFr_Update_DataAxisConfig"(dataAxisConfigLaxisCtrlApcFR := #dataAxisConfig, dataAxisConfigLaxisCtrl => #statDataAxisConfigLAxisCtrl)
   END_RUNG
   // the same network as SCL:
   "LAxisCtrlApcFr_Update_DataAxisConfig"(dataAxisConfigLaxisCtrlApcFR := #dataAxisConfig,
                           dataAxisConfigLaxisCtrl => #statDataAxisConfigLAxisCtrl);
END_REGION

REGION Network 6: (** SELECT CAM **)
   RUNG wire#powerrail
      "LAxisCtrlApcFr_SelectCam"(cam1 := #cam1, camSelection := #dataAxisConfig.camInExtended.camSelection, cam2 := #cam2, TOCam => #statCam, error => #statErrorCamSelection, camSelected => #camSelected)
   END_RUNG
   RUNG wire#powerrail
      "LAxisCtrlApcFr_SelectCam"(cam1 := #cam1, camSelection := #dataAxisConfig.camInStandStill.camSelection, cam2 := #cam2, TOCam => #statCamStandStill, error => #statErrorCamStandStillSelection, camSelected => #statCamStanStillSelected)
   END_RUNG
   // the same network as SCL:
   "LAxisCtrlApcFr_SelectCam"(cam1 := #cam1,
                           camSelection := #dataAxisConfig.camInExtended.camSelection,
                           cam2 := #cam2,
                           TOCam => #statCam,
                           error => #statErrorCamSelection,
                           camSelected => #camSelected);
   "LAxisCtrlApcFr_SelectCam"(cam1 := #cam1,
                           camSelection := #dataAxisConfig.camInStandStill.camSelection,
                           cam2 := #cam2,
                           TOCam => #statCamStandStill,
                           error => #statErrorCamStandStillSelection,
                           camSelected => #statCamStanStillSelected);
END_REGION

REGION Network 7: (** INTERPOLATE CAM **)
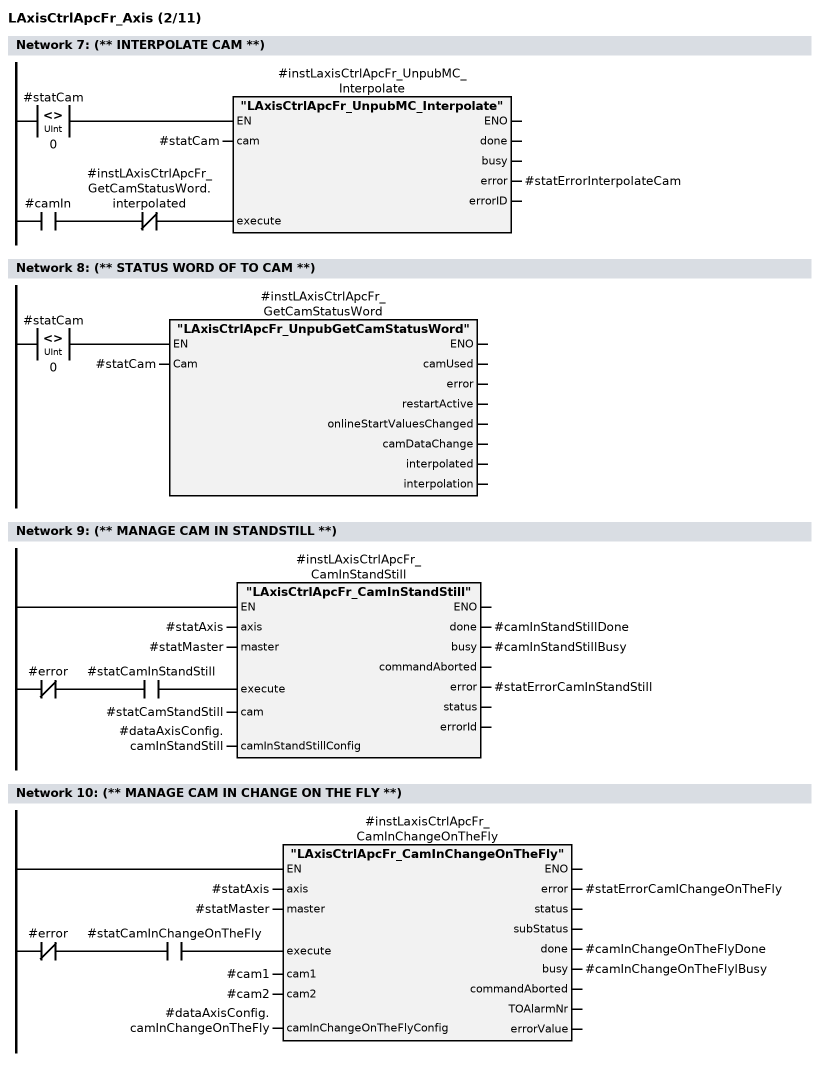
   RUNG wire#powerrail
      { S7_Templates := "SrcType := UInt" } NE_Contact(in1 := #statCam, in2 := 0)
      #instLaxisCtrlApcFr_UnpubMC_Interpolate(execute := wire#w1, cam := #statCam, done =>, busy =>, error => #statErrorInterpolateCam, errorID =>)
   END_RUNG
   RUNG wire#powerrail
      Contact( #camIn )
      I_Contact( #instLAxisCtrlApcFr_GetCamStatusWord.interpolated )
   END_RUNG wire#w1
   // the same network as SCL:
   IF #statCam <> 0 THEN
       #instLaxisCtrlApcFr_UnpubMC_Interpolate(cam := #statCam,   // "LAxisCtrlApcFr_UnpubMC_Interpolate"
                               execute := #camIn AND NOT #instLAxisCtrlApcFr_GetCamStatusWord.interpolated,
                               error => #statErrorInterpolateCam);
   END_IF;
END_REGION

REGION Network 8: (** STATUS WORD OF TO CAM **)
   RUNG wire#powerrail
      { S7_Templates := "SrcType := UInt" } NE_Contact(in1 := #statCam, in2 := 0)
      #instLAxisCtrlApcFr_GetCamStatusWord(Cam := #statCam, camUsed =>, error =>, restartActive =>, onlineStartValuesChanged =>, camDataChange =>, interpolated =>, interpolation =>)
   END_RUNG
   // the same network as SCL:
   IF #statCam <> 0 THEN
       #instLAxisCtrlApcFr_GetCamStatusWord(Cam := #statCam);   // "LAxisCtrlApcFr_UnpubGetCamStatusWord"
   END_IF;
END_REGION

REGION Network 9: (** MANAGE CAM IN STANDSTILL **)
   RUNG wire#powerrail
      #instLAxisCtrlApcFr_CamInStandStill(execute := wire#w1, axis := #statAxis, master := #statMaster, cam := #statCamStandStill, camInStandStillConfig := #dataAxisConfig.camInStandStill, done => #camInStandStillDone, busy => #camInStandStillBusy, commandAborted =>, error => #statErrorCamInStandStill, status =>, errorId =>)
   END_RUNG
   RUNG wire#powerrail
      I_Contact( #error )
      Contact( #statCamInStandStill )
   END_RUNG wire#w1
   // the same network as SCL:
   #instLAxisCtrlApcFr_CamInStandStill(axis := #statAxis,   // "LAxisCtrlApcFr_CamInStandStill"
                           master := #statMaster,
                           execute := NOT #error AND #statCamInStandStill,
                           cam := #statCamStandStill,
                           camInStandStillConfig := #dataAxisConfig.camInStandStill,
                           done => #camInStandStillDone,
                           busy => #camInStandStillBusy,
                           error => #statErrorCamInStandStill);
END_REGION

REGION Network 10: (** MANAGE CAM IN CHANGE ON THE FLY **)
   RUNG wire#powerrail
      #instLaxisCtrlApcFr_CamInChangeOnTheFly(execute := wire#w1, axis := #statAxis, master := #statMaster, cam1 := #cam1, cam2 := #cam2, camInChangeOnTheFlyConfig := #dataAxisConfig.camInChangeOnTheFly, error => #statErrorCamIChangeOnTheFly, status =>, subStatus =>, done => #camInChangeOnTheFlyDone, busy => #camInChangeOnTheFlylBusy, commandAborted =>, TOAlarmNr =>, errorValue =>)
   END_RUNG
   RUNG wire#powerrail
      I_Contact( #error )
      Contact( #statCamInChangeOnTheFly )
   END_RUNG wire#w1
   // the same network as SCL:
   #instLaxisCtrlApcFr_CamInChangeOnTheFly(axis := #statAxis,   // "LAxisCtrlApcFr_CamInChangeOnTheFly"
                           master := #statMaster,
                           execute := NOT #error AND #statCamInChangeOnTheFly,
                           cam1 := #cam1,
                           cam2 := #cam2,
                           camInChangeOnTheFlyConfig := #dataAxisConfig.camInChangeOnTheFly,
                           error => #statErrorCamIChangeOnTheFly,
                           done => #camInChangeOnTheFlyDone,
                           busy => #camInChangeOnTheFlylBusy);
END_REGION

REGION Network 11: (** CALL LAXISCTRL STD SYNC CAMMING **) / (** CALL LAXISCTRL AXIS **)
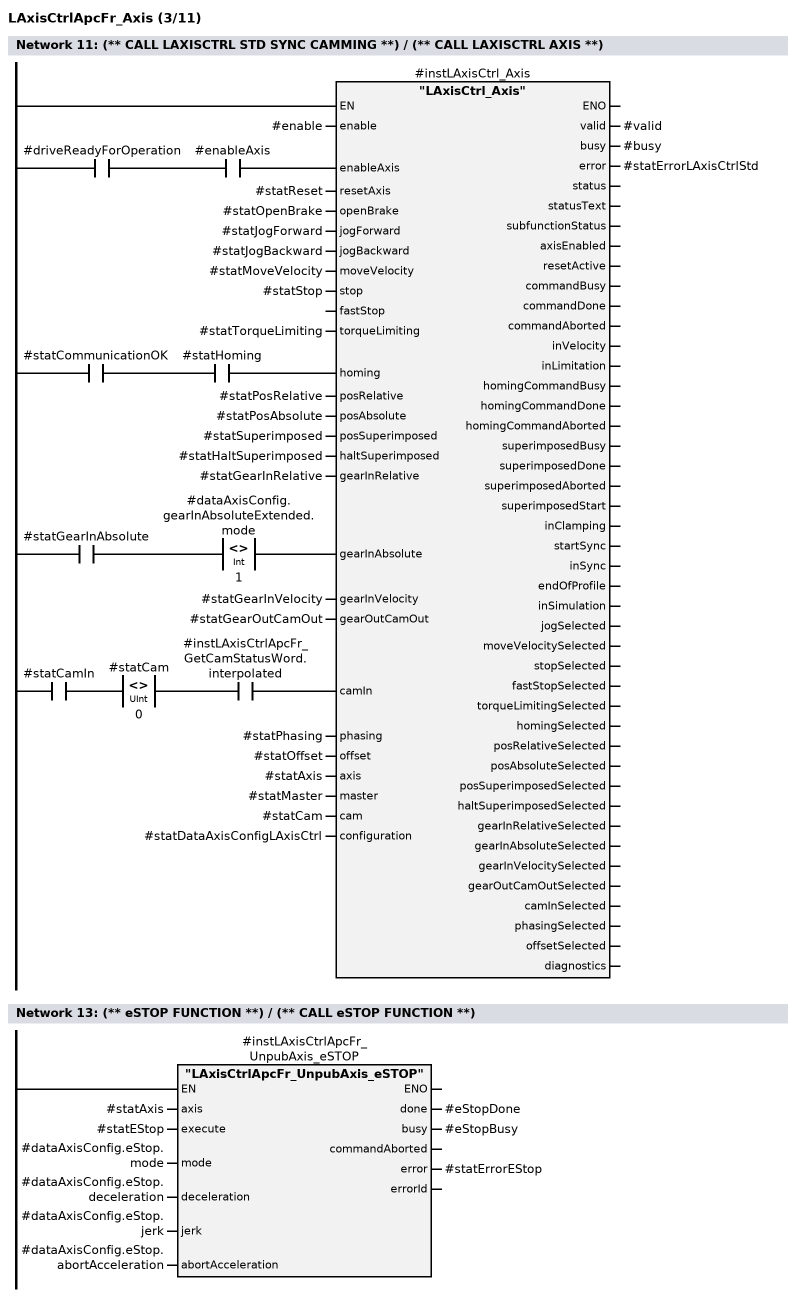
   RUNG wire#powerrail
      #instLAxisCtrl_Axis(enableAxis := wire#w1, homing := wire#w2, gearInAbsolute := wire#w3, camIn := wire#w4, enable := #enable, resetAxis := #statReset, openBrake := #statOpenBrake, jogForward := #statJogForward, jogBackward := #statJogBackward, moveVelocity := #statMoveVelocity, stop := #statStop, fastStop :=, torqueLimiting := #statTorqueLimiting, posRelative := #statPosRelative, posAbsolute := #statPosAbsolute, posSuperimposed := #statSuperimposed, haltSuperimposed := #statHaltSuperimposed, gearInRelative := #statGearInRelative, gearInVelocity := #statGearInVelocity, gearOutCamOut := #statGearOutCamOut, phasing := #statPhasing, offset := #statOffset, axis := #statAxis, master := #statMaster, cam := #statCam, configuration := #statDataAxisConfigLAxisCtrl, valid => #valid, busy => #busy, error => #statErrorLAxisCtrlStd, status =>, statusText =>, subfunctionStatus =>, axisEnabled =>, resetActive =>, commandBusy =>, commandDone =>, commandAborted =>, inVelocity =>, inLimitation =>, homingCommandBusy =>, homingCommandDone =>, homingCommandAborted =>, superimposedBusy =>, superimposedDone =>, superimposedAborted =>, superimposedStart =>, inClamping =>, startSync =>, inSync =>, endOfProfile =>, inSimulation =>, jogSelected =>, moveVelocitySelected =>, stopSelected =>, fastStopSelected =>, torqueLimitingSelected =>, homingSelected =>, posRelativeSelected =>, posAbsoluteSelected =>, posSuperimposedSelected =>, haltSuperimposedSelected =>, gearInRelativeSelected =>, gearInAbsoluteSelected =>, gearInVelocitySelected =>, gearOutCamOutSelected =>, camInSelected =>, phasingSelected =>, offsetSelected =>, diagnostics =>)
   END_RUNG
   RUNG wire#powerrail
      Contact( #driveReadyForOperation )
      Contact( #enableAxis )
   END_RUNG wire#w1
   RUNG wire#powerrail
      Contact( #statCommunicationOK )
      Contact( #statHoming )
   END_RUNG wire#w2
   RUNG wire#powerrail
      Contact( #statGearInAbsolute )
      { S7_Templates := "SrcType := Int" } NE_Contact(in1 := #dataAxisConfig.gearInAbsoluteExtended.mode, in2 := 1)
   END_RUNG wire#w3
   RUNG wire#powerrail
      Contact( #statCamIn )
      { S7_Templates := "SrcType := UInt" } NE_Contact(in1 := #statCam, in2 := 0)
      Contact( #instLAxisCtrlApcFr_GetCamStatusWord.interpolated )
   END_RUNG wire#w4
   // the same network as SCL:
   #instLAxisCtrl_Axis(enable := #enable,   // "LAxisCtrl_Axis"
                       enableAxis := #driveReadyForOperation AND #enableAxis,
                       resetAxis := #statReset,
                       openBrake := #statOpenBrake,
                       jogForward := #statJogForward,
                       jogBackward := #statJogBackward,
                       moveVelocity := #statMoveVelocity,
                       stop := #statStop,
                       torqueLimiting := #statTorqueLimiting,
                       homing := #statCommunicationOK AND #statHoming,
                       posRelative := #statPosRelative,
                       posAbsolute := #statPosAbsolute,
                       posSuperimposed := #statSuperimposed,
                       haltSuperimposed := #statHaltSuperimposed,
                       gearInRelative := #statGearInRelative,
                       gearInAbsolute := #statGearInAbsolute AND (#dataAxisConfig.gearInAbsoluteExtended.mode <> 1),
                       gearInVelocity := #statGearInVelocity,
                       gearOutCamOut := #statGearOutCamOut,
                       camIn := #statCamIn AND (#statCam <> 0) AND #instLAxisCtrlApcFr_GetCamStatusWord.interpolated,
                       phasing := #statPhasing,
                       offset := #statOffset,
                       axis := #statAxis,
                       master := #statMaster,
                       cam := #statCam,
                       configuration := #statDataAxisConfigLAxisCtrl,
                       valid => #valid,
                       busy => #busy,
                       error => #statErrorLAxisCtrlStd);
END_REGION

REGION Network 12 (SCL): (** UPDATE OUTPUTS FROM LAXISCTRL STD **)
   #outputsLAxisCtrl_Axis.valid := #instLAxisCtrl_Axis.valid;
   #outputsLAxisCtrl_Axis.busy := #instLAxisCtrl_Axis.busy;
   #outputsLAxisCtrl_Axis.error := #instLAxisCtrl_Axis.error;
   #outputsLAxisCtrl_Axis.status := #instLAxisCtrl_Axis.status;
   #outputsLAxisCtrl_Axis.statusText := #instLAxisCtrl_Axis.statusText;
   #outputsLAxisCtrl_Axis.subfunctionStatus := #instLAxisCtrl_Axis.subfunctionStatus;
   #outputsLAxisCtrl_Axis.axisEnabled := #instLAxisCtrl_Axis.axisEnabled;
   #outputsLAxisCtrl_Axis.resetActive := #instLAxisCtrl_Axis.resetActive;
   #outputsLAxisCtrl_Axis.commandDone := #instLAxisCtrl_Axis.commandDone;
   #outputsLAxisCtrl_Axis.commandAborted := #instLAxisCtrl_Axis.commandAborted;
   #outputsLAxisCtrl_Axis.inVelocity := #instLAxisCtrl_Axis.inVelocity;
   #outputsLAxisCtrl_Axis.inLimitation := #instLAxisCtrl_Axis.inLimitation;
   #outputsLAxisCtrl_Axis.homingCommandBusy := #instLAxisCtrl_Axis.homingCommandBusy;
   #outputsLAxisCtrl_Axis.homingCommandDone := #instLAxisCtrl_Axis.homingCommandDone;
   #outputsLAxisCtrl_Axis.homingCommandAborted := #instLAxisCtrl_Axis.homingCommandAborted;
   #outputsLAxisCtrl_Axis.superimposedBusy := #instLAxisCtrl_Axis.superimposedBusy;
   #outputsLAxisCtrl_Axis.superimposedDone := #instLAxisCtrl_Axis.superimposedDone;
   #outputsLAxisCtrl_Axis.superimposedAborted := #instLAxisCtrl_Axis.superimposedAborted;
   #outputsLAxisCtrl_Axis.superimposedStart := #instLAxisCtrl_Axis.superimposedStart;
   #outputsLAxisCtrl_Axis.inClamping := #instLAxisCtrl_Axis.inClamping;
   #outputsLAxisCtrl_Axis.startSync := #instLAxisCtrl_Axis.startSync;
   #outputsLAxisCtrl_Axis.inSync := #instLAxisCtrl_Axis.inSync;
   #outputsLAxisCtrl_Axis.endOfProfile := #instLAxisCtrl_Axis.endOfProfile;
   #outputsLAxisCtrl_Axis.inSimulation := #instLAxisCtrl_Axis.inSimulation;
   #outputsLAxisCtrl_Axis.jogSelected := #instLAxisCtrl_Axis.jogSelected;
   #outputsLAxisCtrl_Axis.moveVelocitySelected := #instLAxisCtrl_Axis.moveVelocitySelected;
   #outputsLAxisCtrl_Axis.stopSelected := #instLAxisCtrl_Axis.stopSelected;
   #outputsLAxisCtrl_Axis.fastStopSelected := #instLAxisCtrl_Axis.fastStopSelected;
   #outputsLAxisCtrl_Axis.torqueLimitingSelected := #instLAxisCtrl_Axis.torqueLimitingSelected;
   #outputsLAxisCtrl_Axis.homingSelected := #instLAxisCtrl_Axis.homingSelected;
   #outputsLAxisCtrl_Axis.posRelativeSelected := #instLAxisCtrl_Axis.posRelativeSelected;
   #outputsLAxisCtrl_Axis.posAbsoluteSelected := #instLAxisCtrl_Axis.posAbsoluteSelected;
   #outputsLAxisCtrl_Axis.posSuperimposedSelected := #instLAxisCtrl_Axis.posSuperimposedSelected;
   #outputsLAxisCtrl_Axis.haltSuperimposedSelected := #instLAxisCtrl_Axis.haltSuperimposedSelected;
   #outputsLAxisCtrl_Axis.gearInRelativeSelected := #instLAxisCtrl_Axis.gearInRelativeSelected;
   #outputsLAxisCtrl_Axis.gearInAbsoluteSelected := #instLAxisCtrl_Axis.gearInAbsoluteSelected;
   #outputsLAxisCtrl_Axis.gearInVelocitySelected := #instLAxisCtrl_Axis.gearInVelocitySelected;
   #outputsLAxisCtrl_Axis.gearOutCamOutSelected := #instLAxisCtrl_Axis.gearOutCamOutSelected;
   #outputsLAxisCtrl_Axis.camInSelected := #instLAxisCtrl_Axis.camInSelected;
   #outputsLAxisCtrl_Axis.phasingSelected := #instLAxisCtrl_Axis.phasingSelected;
   #outputsLAxisCtrl_Axis.offsetSelected := #instLAxisCtrl_Axis.offsetSelected;
   #outputsLAxisCtrl_Axis.diagnostics := #instLAxisCtrl_Axis.diagnostics;
END_REGION

REGION Network 13: (** eSTOP FUNCTION **) / (** CALL eSTOP FUNCTION **)
   RUNG wire#powerrail
      #instLAxisCtrlApcFr_UnpubAxis_eSTOP(axis := #statAxis, execute := #statEStop, mode := #dataAxisConfig.eStop.mode, deceleration := #dataAxisConfig.eStop.deceleration, jerk := #dataAxisConfig.eStop.jerk, abortAcceleration := #dataAxisConfig.eStop.abortAcceleration, done => #eStopDone, busy => #eStopBusy, commandAborted =>, error => #statErrorEStop, errorId =>)
   END_RUNG
   // the same network as SCL:
   #instLAxisCtrlApcFr_UnpubAxis_eSTOP(axis := #statAxis,   // "LAxisCtrlApcFr_UnpubAxis_eSTOP"
                           execute := #statEStop,
                           mode := #dataAxisConfig.eStop.mode,
                           deceleration := #dataAxisConfig.eStop.deceleration,
                           jerk := #dataAxisConfig.eStop.jerk,
                           abortAcceleration := #dataAxisConfig.eStop.abortAcceleration,
                           done => #eStopDone,
                           busy => #eStopBusy,
                           error => #statErrorEStop);
END_REGION

REGION Network 14: (** CALL GEARINPOS **)
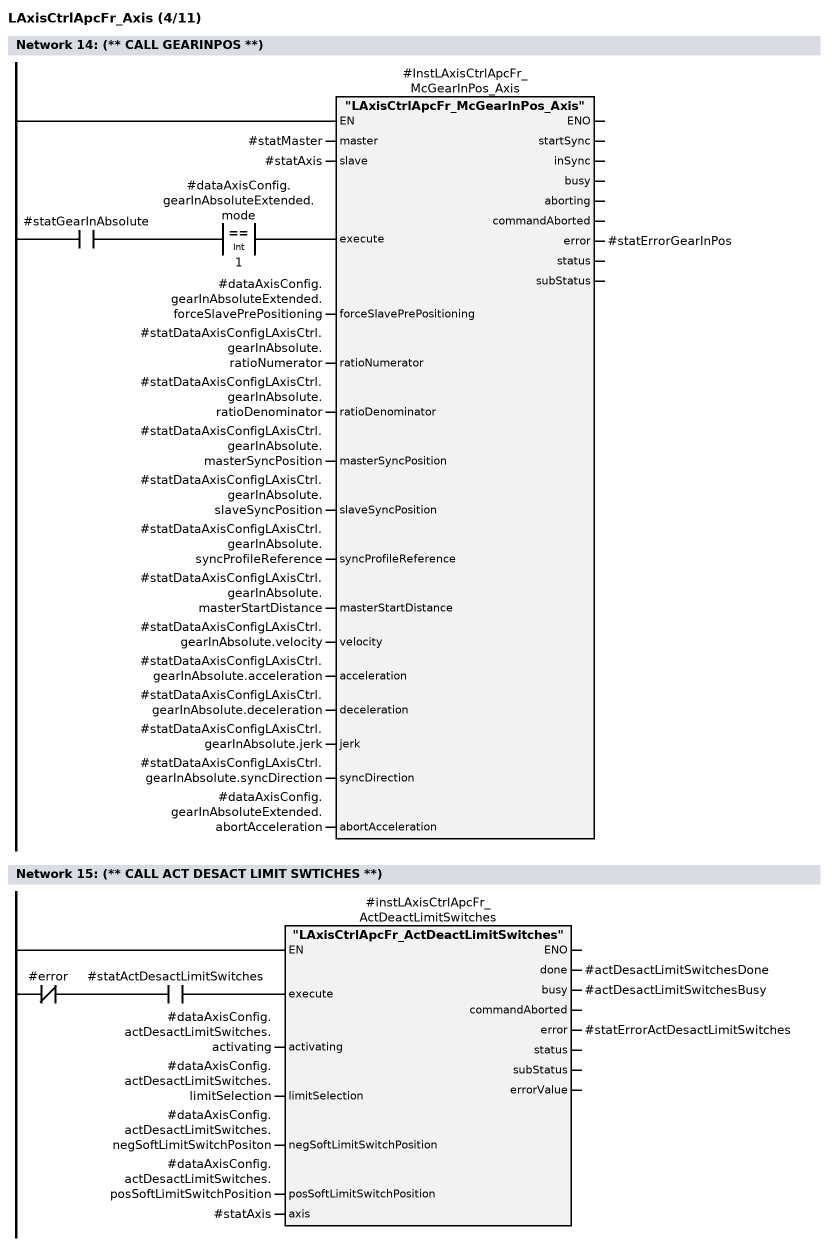
   RUNG wire#powerrail
      #InstLAxisCtrlApcFr_McGearInPos_Axis(execute := wire#w1, master := #statMaster, slave := #statAxis, forceSlavePrePositioning := #dataAxisConfig.gearInAbsoluteExtended.forceSlavePrePositioning, ratioNumerator := #statDataAxisConfigLAxisCtrl.gearInAbsolute.ratioNumerator, ratioDenominator := #statDataAxisConfigLAxisCtrl.gearInAbsolute.ratioDenominator, masterSyncPosition := #statDataAxisConfigLAxisCtrl.gearInAbsolute.masterSyncPosition, slaveSyncPosition := #statDataAxisConfigLAxisCtrl.gearInAbsolute.slaveSyncPosition, syncProfileReference := #statDataAxisConfigLAxisCtrl.gearInAbsolute.syncProfileReference, masterStartDistance := #statDataAxisConfigLAxisCtrl.gearInAbsolute.masterStartDistance, velocity := #statDataAxisConfigLAxisCtrl.gearInAbsolute.velocity, acceleration := #statDataAxisConfigLAxisCtrl.gearInAbsolute.acceleration, deceleration := #statDataAxisConfigLAxisCtrl.gearInAbsolute.deceleration, jerk := #statDataAxisConfigLAxisCtrl.gearInAbsolute.jerk, syncDirection := #statDataAxisConfigLAxisCtrl.gearInAbsolute.syncDirection, abortAcceleration := #dataAxisConfig.gearInAbsoluteExtended.abortAcceleration, startSync =>, inSync =>, busy =>, aborting =>, commandAborted =>, error => #statErrorGearInPos, status =>, subStatus =>)
   END_RUNG
   RUNG wire#powerrail
      Contact( #statGearInAbsolute )
      { S7_Templates := "SrcType := Int" } EQ_Contact(in1 := #dataAxisConfig.gearInAbsoluteExtended.mode, in2 := 1)
   END_RUNG wire#w1
   // the same network as SCL:
   #InstLAxisCtrlApcFr_McGearInPos_Axis(master := #statMaster,   // "LAxisCtrlApcFr_McGearInPos_Axis"
                           slave := #statAxis,
                           execute := #statGearInAbsolute AND (#dataAxisConfig.gearInAbsoluteExtended.mode = 1),
                           forceSlavePrePositioning := #dataAxisConfig.gearInAbsoluteExtended.forceSlavePrePositioning,
                           ratioNumerator := #statDataAxisConfigLAxisCtrl.gearInAbsolute.ratioNumerator,
                           ratioDenominator := #statDataAxisConfigLAxisCtrl.gearInAbsolute.ratioDenominator,
                           masterSyncPosition := #statDataAxisConfigLAxisCtrl.gearInAbsolute.masterSyncPosition,
                           slaveSyncPosition := #statDataAxisConfigLAxisCtrl.gearInAbsolute.slaveSyncPosition,
                           syncProfileReference := #statDataAxisConfigLAxisCtrl.gearInAbsolute.syncProfileReference,
                           masterStartDistance := #statDataAxisConfigLAxisCtrl.gearInAbsolute.masterStartDistance,
                           velocity := #statDataAxisConfigLAxisCtrl.gearInAbsolute.velocity,
                           acceleration := #statDataAxisConfigLAxisCtrl.gearInAbsolute.acceleration,
                           deceleration := #statDataAxisConfigLAxisCtrl.gearInAbsolute.deceleration,
                           jerk := #statDataAxisConfigLAxisCtrl.gearInAbsolute.jerk,
                           syncDirection := #statDataAxisConfigLAxisCtrl.gearInAbsolute.syncDirection,
                           abortAcceleration := #dataAxisConfig.gearInAbsoluteExtended.abortAcceleration,
                           error => #statErrorGearInPos);
END_REGION

REGION Network 15: (** CALL ACT DESACT LIMIT SWTICHES **)
   RUNG wire#powerrail
      #instLAxisCtrlApcFr_ActDeactLimitSwitches(execute := wire#w1, activating := #dataAxisConfig.actDesactLimitSwitches.activating, limitSelection := #dataAxisConfig.actDesactLimitSwitches.limitSelection, negSoftLimitSwitchPosition := #dataAxisConfig.actDesactLimitSwitches.negSoftLimitSwitchPositon, posSoftLimitSwitchPosition := #dataAxisConfig.actDesactLimitSwitches.posSoftLimitSwitchPosition, axis := #statAxis, done => #actDesactLimitSwitchesDone, busy => #actDesactLimitSwitchesBusy, commandAborted =>, error => #statErrorActDesactLimitSwitches, status =>, subStatus =>, errorValue =>)
   END_RUNG
   RUNG wire#powerrail
      I_Contact( #error )
      Contact( #statActDesactLimitSwitches )
   END_RUNG wire#w1
   // the same network as SCL:
   #instLAxisCtrlApcFr_ActDeactLimitSwitches(execute := NOT #error AND #statActDesactLimitSwitches,   // "LAxisCtrlApcFr_ActDeactLimitSwitches"
                           activating := #dataAxisConfig.actDesactLimitSwitches.activating,
                           limitSelection := #dataAxisConfig.actDesactLimitSwitches.limitSelection,
                           negSoftLimitSwitchPosition := #dataAxisConfig.actDesactLimitSwitches.negSoftLimitSwitchPositon,
                           posSoftLimitSwitchPosition := #dataAxisConfig.actDesactLimitSwitches.posSoftLimitSwitchPosition,
                           axis := #statAxis,
                           done => #actDesactLimitSwitchesDone,
                           busy => #actDesactLimitSwitchesBusy,
                           error => #statErrorActDesactLimitSwitches);
END_REGION

REGION Network 16: (** CALL CHANGE MODULO AXIS **)
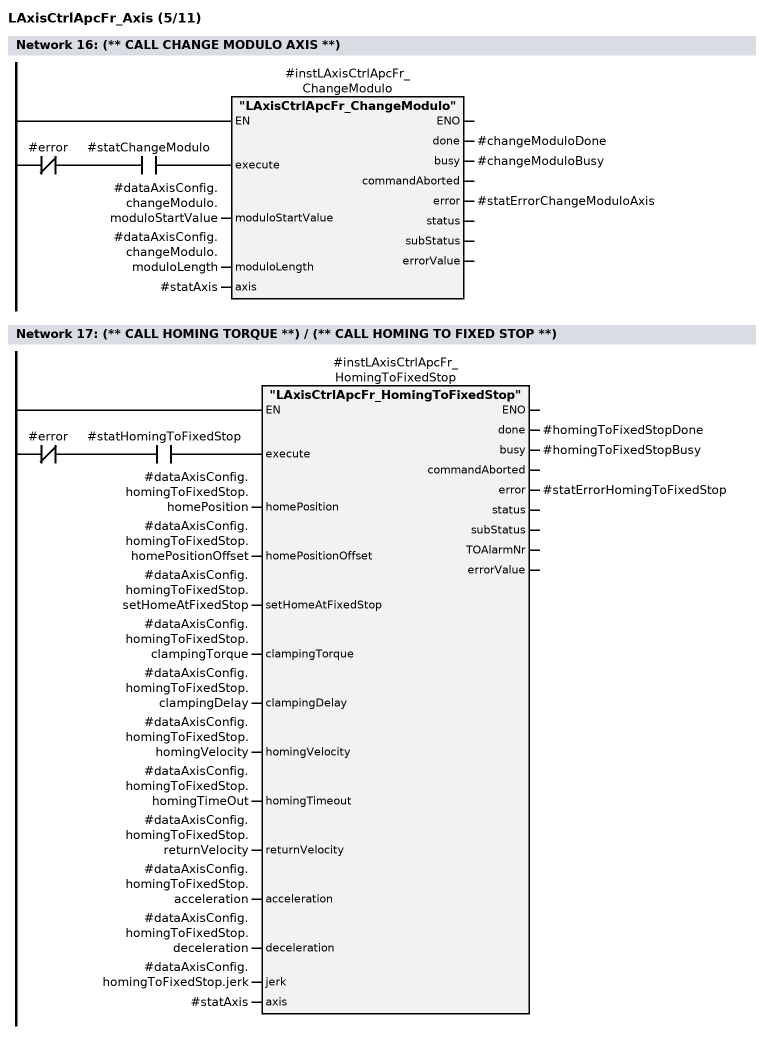
   RUNG wire#powerrail
      #instLAxisCtrlApcFr_ChangeModulo(execute := wire#w1, moduloStartValue := #dataAxisConfig.changeModulo.moduloStartValue, moduloLength := #dataAxisConfig.changeModulo.moduloLength, axis := #statAxis, done => #changeModuloDone, busy => #changeModuloBusy, commandAborted =>, error => #statErrorChangeModuloAxis, status =>, subStatus =>, errorValue =>)
   END_RUNG
   RUNG wire#powerrail
      I_Contact( #error )
      Contact( #statChangeModulo )
   END_RUNG wire#w1
   // the same network as SCL:
   #instLAxisCtrlApcFr_ChangeModulo(execute := NOT #error AND #statChangeModulo,   // "LAxisCtrlApcFr_ChangeModulo"
                           moduloStartValue := #dataAxisConfig.changeModulo.moduloStartValue,
                           moduloLength := #dataAxisConfig.changeModulo.moduloLength,
                           axis := #statAxis,
                           done => #changeModuloDone,
                           busy => #changeModuloBusy,
                           error => #statErrorChangeModuloAxis);
END_REGION

REGION Network 17: (** CALL HOMING TORQUE **) / (** CALL HOMING TO FIXED STOP **)
   RUNG wire#powerrail
      #instLAxisCtrlApcFr_HomingToFixedStop(execute := wire#w1, homePosition := #dataAxisConfig.homingToFixedStop.homePosition, homePositionOffset := #dataAxisConfig.homingToFixedStop.homePositionOffset, setHomeAtFixedStop := #dataAxisConfig.homingToFixedStop.setHomeAtFixedStop, clampingTorque := #dataAxisConfig.homingToFixedStop.clampingTorque, clampingDelay := #dataAxisConfig.homingToFixedStop.clampingDelay, homingVelocity := #dataAxisConfig.homingToFixedStop.homingVelocity, homingTimeout := #dataAxisConfig.homingToFixedStop.homingTimeOut, returnVelocity := #dataAxisConfig.homingToFixedStop.returnVelocity, acceleration := #dataAxisConfig.homingToFixedStop.acceleration, deceleration := #dataAxisConfig.homingToFixedStop.deceleration, jerk := #dataAxisConfig.homingToFixedStop.jerk, axis := #statAxis, done => #homingToFixedStopDone, busy => #homingToFixedStopBusy, commandAborted =>, error => #statErrorHomingToFixedStop, status =>, subStatus =>, TOAlarmNr =>, errorValue =>)
   END_RUNG
   RUNG wire#powerrail
      I_Contact( #error )
      Contact( #statHomingToFixedStop )
   END_RUNG wire#w1
   // the same network as SCL:
   #instLAxisCtrlApcFr_HomingToFixedStop(execute := NOT #error AND #statHomingToFixedStop,   // "LAxisCtrlApcFr_HomingToFixedStop"
                           homePosition := #dataAxisConfig.homingToFixedStop.homePosition,
                           homePositionOffset := #dataAxisConfig.homingToFixedStop.homePositionOffset,
                           setHomeAtFixedStop := #dataAxisConfig.homingToFixedStop.setHomeAtFixedStop,
                           clampingTorque := #dataAxisConfig.homingToFixedStop.clampingTorque,
                           clampingDelay := #dataAxisConfig.homingToFixedStop.clampingDelay,
                           homingVelocity := #dataAxisConfig.homingToFixedStop.homingVelocity,
                           homingTimeout := #dataAxisConfig.homingToFixedStop.homingTimeOut,
                           returnVelocity := #dataAxisConfig.homingToFixedStop.returnVelocity,
                           acceleration := #dataAxisConfig.homingToFixedStop.acceleration,
                           deceleration := #dataAxisConfig.homingToFixedStop.deceleration,
                           jerk := #dataAxisConfig.homingToFixedStop.jerk,
                           axis := #statAxis,
                           done => #homingToFixedStopDone,
                           busy => #homingToFixedStopBusy,
                           error => #statErrorHomingToFixedStop);
END_REGION

REGION Network 18: (** CALL HOMING ON SENSOR **)
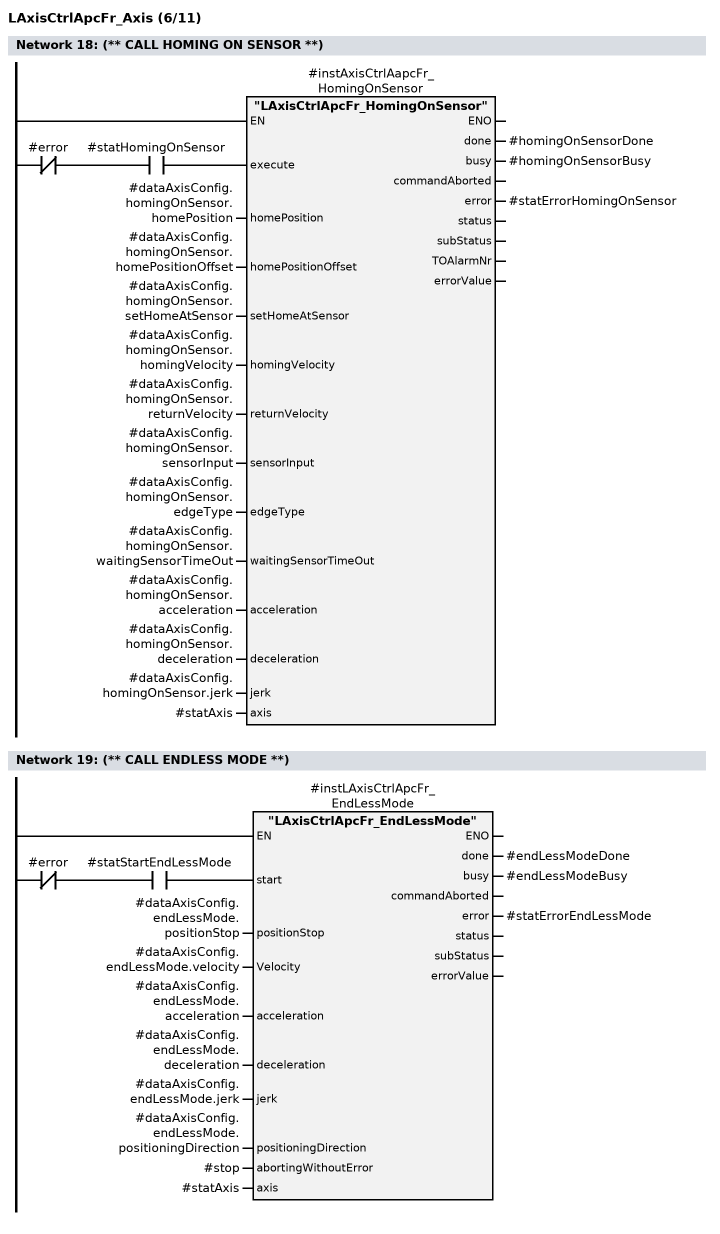
   RUNG wire#powerrail
      #instAxisCtrlAapcFr_HomingOnSensor(execute := wire#w1, homePosition := #dataAxisConfig.homingOnSensor.homePosition, homePositionOffset := #dataAxisConfig.homingOnSensor.homePositionOffset, setHomeAtSensor := #dataAxisConfig.homingOnSensor.setHomeAtSensor, homingVelocity := #dataAxisConfig.homingOnSensor.homingVelocity, returnVelocity := #dataAxisConfig.homingOnSensor.returnVelocity, sensorInput := #dataAxisConfig.homingOnSensor.sensorInput, edgeType := #dataAxisConfig.homingOnSensor.edgeType, waitingSensorTimeOut := #dataAxisConfig.homingOnSensor.waitingSensorTimeOut, acceleration := #dataAxisConfig.homingOnSensor.acceleration, deceleration := #dataAxisConfig.homingOnSensor.deceleration, jerk := #dataAxisConfig.homingOnSensor.jerk, axis := #statAxis, done => #homingOnSensorDone, busy => #homingOnSensorBusy, commandAborted =>, error => #statErrorHomingOnSensor, status =>, subStatus =>, TOAlarmNr =>, errorValue =>)
   END_RUNG
   RUNG wire#powerrail
      I_Contact( #error )
      Contact( #statHomingOnSensor )
   END_RUNG wire#w1
   // the same network as SCL:
   #instAxisCtrlAapcFr_HomingOnSensor(execute := NOT #error AND #statHomingOnSensor,   // "LAxisCtrlApcFr_HomingOnSensor"
                           homePosition := #dataAxisConfig.homingOnSensor.homePosition,
                           homePositionOffset := #dataAxisConfig.homingOnSensor.homePositionOffset,
                           setHomeAtSensor := #dataAxisConfig.homingOnSensor.setHomeAtSensor,
                           homingVelocity := #dataAxisConfig.homingOnSensor.homingVelocity,
                           returnVelocity := #dataAxisConfig.homingOnSensor.returnVelocity,
                           sensorInput := #dataAxisConfig.homingOnSensor.sensorInput,
                           edgeType := #dataAxisConfig.homingOnSensor.edgeType,
                           waitingSensorTimeOut := #dataAxisConfig.homingOnSensor.waitingSensorTimeOut,
                           acceleration := #dataAxisConfig.homingOnSensor.acceleration,
                           deceleration := #dataAxisConfig.homingOnSensor.deceleration,
                           jerk := #dataAxisConfig.homingOnSensor.jerk,
                           axis := #statAxis,
                           done => #homingOnSensorDone,
                           busy => #homingOnSensorBusy,
                           error => #statErrorHomingOnSensor);
END_REGION

REGION Network 19: (** CALL ENDLESS MODE **)
   RUNG wire#powerrail
      #instLAxisCtrlApcFr_EndLessMode(start := wire#w1, positionStop := #dataAxisConfig.endLessMode.positionStop, Velocity := #dataAxisConfig.endLessMode.velocity, acceleration := #dataAxisConfig.endLessMode.acceleration, deceleration := #dataAxisConfig.endLessMode.deceleration, jerk := #dataAxisConfig.endLessMode.jerk, positioningDirection := #dataAxisConfig.endLessMode.positioningDirection, abortingWithoutError := #stop, axis := #statAxis, done => #endLessModeDone, busy => #endLessModeBusy, commandAborted =>, error => #statErrorEndLessMode, status =>, subStatus =>, errorValue =>)
   END_RUNG
   RUNG wire#powerrail
      I_Contact( #error )
      Contact( #statStartEndLessMode )
   END_RUNG wire#w1
   // the same network as SCL:
   #instLAxisCtrlApcFr_EndLessMode(start := NOT #error AND #statStartEndLessMode,   // "LAxisCtrlApcFr_EndLessMode"
                           positionStop := #dataAxisConfig.endLessMode.positionStop,
                           Velocity := #dataAxisConfig.endLessMode.velocity,
                           acceleration := #dataAxisConfig.endLessMode.acceleration,
                           deceleration := #dataAxisConfig.endLessMode.deceleration,
                           jerk := #dataAxisConfig.endLessMode.jerk,
                           positioningDirection := #dataAxisConfig.endLessMode.positioningDirection,
                           abortingWithoutError := #stop,
                           axis := #statAxis,
                           done => #endLessModeDone,
                           busy => #endLessModeBusy,
                           error => #statErrorEndLessMode);
END_REGION

REGION Network 20: (** CALL SIMULATION ON OFF **)
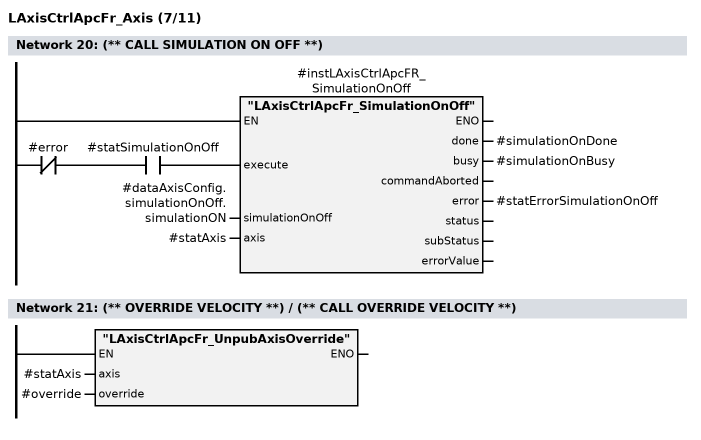
   RUNG wire#powerrail
      #instLAxisCtrlApcFR_SimulationOnOff(execute := wire#w1, simulationOnOff := #dataAxisConfig.simulationOnOff.simulationON, axis := #statAxis, done => #simulationOnDone, busy => #simulationOnBusy, commandAborted =>, error => #statErrorSimulationOnOff, status =>, subStatus =>, errorValue =>)
   END_RUNG
   RUNG wire#powerrail
      I_Contact( #error )
      Contact( #statSimulationOnOff )
   END_RUNG wire#w1
   // the same network as SCL:
   #instLAxisCtrlApcFR_SimulationOnOff(execute := NOT #error AND #statSimulationOnOff,   // "LAxisCtrlApcFr_SimulationOnOff"
                           simulationOnOff := #dataAxisConfig.simulationOnOff.simulationON,
                           axis := #statAxis,
                           done => #simulationOnDone,
                           busy => #simulationOnBusy,
                           error => #statErrorSimulationOnOff);
END_REGION

REGION Network 21: (** OVERRIDE VELOCITY **) / (** CALL OVERRIDE VELOCITY **)
   RUNG wire#powerrail
      "LAxisCtrlApcFr_UnpubAxisOverride"(axis := #statAxis, override := #override)
   END_RUNG
   // the same network as SCL:
   "LAxisCtrlApcFr_UnpubAxisOverride"(axis := #statAxis, override := #override);
END_REGION

REGION Network 22: (** STATUS WORD OF TO AXIS **)
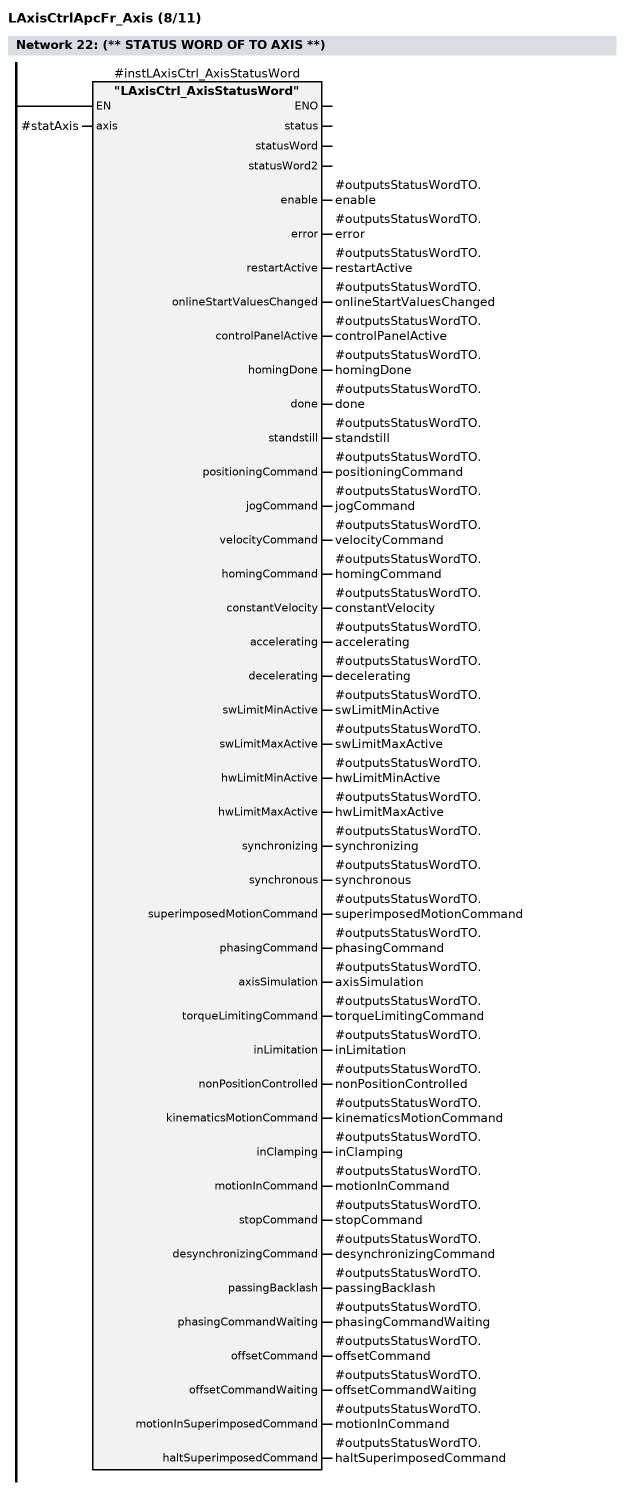
   RUNG wire#powerrail
      #instLAxisCtrl_AxisStatusWord(axis := #statAxis, status =>, statusWord =>, statusWord2 =>, enable => #outputsStatusWordTO.enable, error => #outputsStatusWordTO.error, restartActive => #outputsStatusWordTO.restartActive, onlineStartValuesChanged => #outputsStatusWordTO.onlineStartValuesChanged, controlPanelActive => #outputsStatusWordTO.controlPanelActive, homingDone => #outputsStatusWordTO.homingDone, done => #outputsStatusWordTO.done, standstill => #outputsStatusWordTO.standstill, positioningCommand => #outputsStatusWordTO.positioningCommand, jogCommand => #outputsStatusWordTO.jogCommand, velocityCommand => #outputsStatusWordTO.velocityCommand, homingCommand => #outputsStatusWordTO.homingCommand, constantVelocity => #outputsStatusWordTO.constantVelocity, accelerating => #outputsStatusWordTO.accelerating, decelerating => #outputsStatusWordTO.decelerating, swLimitMinActive => #outputsStatusWordTO.swLimitMinActive, swLimitMaxActive => #outputsStatusWordTO.swLimitMaxActive, hwLimitMinActive => #outputsStatusWordTO.hwLimitMinActive, hwLimitMaxActive => #outputsStatusWordTO.hwLimitMaxActive, synchronizing => #outputsStatusWordTO.synchronizing, synchronous => #outputsStatusWordTO.synchronous, superimposedMotionCommand => #outputsStatusWordTO.superimposedMotionCommand, phasingCommand => #outputsStatusWordTO.phasingCommand, axisSimulation => #outputsStatusWordTO.axisSimulation, torqueLimitingCommand => #outputsStatusWordTO.torqueLimitingCommand, inLimitation => #outputsStatusWordTO.inLimitation, nonPositionControlled => #outputsStatusWordTO.nonPositionControlled, kinematicsMotionCommand => #outputsStatusWordTO.kinematicsMotionCommand, inClamping => #outputsStatusWordTO.inClamping, motionInCommand => #outputsStatusWordTO.motionInCommand, stopCommand => #outputsStatusWordTO.stopCommand, desynchronizingCommand => #outputsStatusWordTO.desynchronizingCommand, passingBacklash => #outputsStatusWordTO.passingBacklash, phasingCommandWaiting => #outputsStatusWordTO.phasingCommandWaiting, offsetCommand => #outputsStatusWordTO.offsetCommand, offsetCommandWaiting => #outputsStatusWordTO.offsetCommandWaiting, motionInSuperimposedCommand => #outputsStatusWordTO.motionInCommand, haltSuperimposedCommand => #outputsStatusWordTO.haltSuperimposedCommand)
   END_RUNG
   // the same network as SCL:
   #instLAxisCtrl_AxisStatusWord(axis := #statAxis,   // "LAxisCtrl_AxisStatusWord"
                           enable => #outputsStatusWordTO.enable,
                           error => #outputsStatusWordTO.error,
                           restartActive => #outputsStatusWordTO.restartActive,
                           onlineStartValuesChanged => #outputsStatusWordTO.onlineStartValuesChanged,
                           controlPanelActive => #outputsStatusWordTO.controlPanelActive,
                           homingDone => #outputsStatusWordTO.homingDone,
                           done => #outputsStatusWordTO.done,
                           standstill => #outputsStatusWordTO.standstill,
                           positioningCommand => #outputsStatusWordTO.positioningCommand,
                           jogCommand => #outputsStatusWordTO.jogCommand,
                           velocityCommand => #outputsStatusWordTO.velocityCommand,
                           homingCommand => #outputsStatusWordTO.homingCommand,
                           constantVelocity => #outputsStatusWordTO.constantVelocity,
                           accelerating => #outputsStatusWordTO.accelerating,
                           decelerating => #outputsStatusWordTO.decelerating,
                           swLimitMinActive => #outputsStatusWordTO.swLimitMinActive,
                           swLimitMaxActive => #outputsStatusWordTO.swLimitMaxActive,
                           hwLimitMinActive => #outputsStatusWordTO.hwLimitMinActive,
                           hwLimitMaxActive => #outputsStatusWordTO.hwLimitMaxActive,
                           synchronizing => #outputsStatusWordTO.synchronizing,
                           synchronous => #outputsStatusWordTO.synchronous,
                           superimposedMotionCommand => #outputsStatusWordTO.superimposedMotionCommand,
                           phasingCommand => #outputsStatusWordTO.phasingCommand,
                           axisSimulation => #outputsStatusWordTO.axisSimulation,
                           torqueLimitingCommand => #outputsStatusWordTO.torqueLimitingCommand,
                           inLimitation => #outputsStatusWordTO.inLimitation,
                           nonPositionControlled => #outputsStatusWordTO.nonPositionControlled,
                           kinematicsMotionCommand => #outputsStatusWordTO.kinematicsMotionCommand,
                           inClamping => #outputsStatusWordTO.inClamping,
                           motionInCommand => #outputsStatusWordTO.motionInCommand,
                           stopCommand => #outputsStatusWordTO.stopCommand,
                           desynchronizingCommand => #outputsStatusWordTO.desynchronizingCommand,
                           passingBacklash => #outputsStatusWordTO.passingBacklash,
                           phasingCommandWaiting => #outputsStatusWordTO.phasingCommandWaiting,
                           offsetCommand => #outputsStatusWordTO.offsetCommand,
                           offsetCommandWaiting => #outputsStatusWordTO.offsetCommandWaiting,
                           motionInSuperimposedCommand => #outputsStatusWordTO.motionInCommand,
                           haltSuperimposedCommand => #outputsStatusWordTO.haltSuperimposedCommand);
END_REGION

REGION Network 23: (** STATUS DWORD OF AXIS COMMAND **)
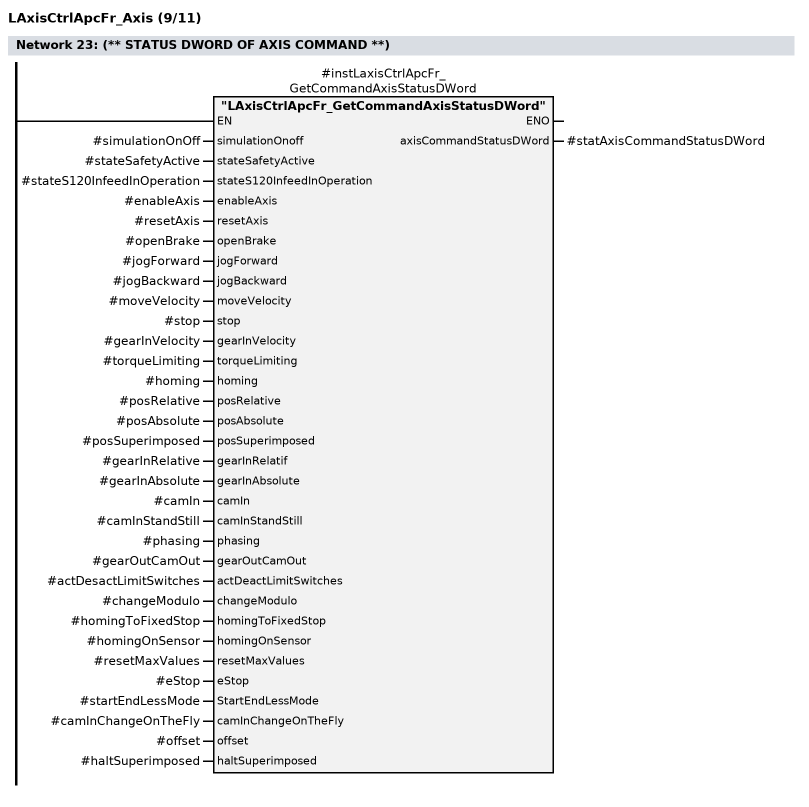
   RUNG wire#powerrail
      #instLaxisCtrlApcFr_GetCommandAxisStatusDWord(simulationOnoff := #simulationOnOff, stateSafetyActive := #stateSafetyActive, stateS120InfeedInOperation := #stateS120InfeedInOperation, enableAxis := #enableAxis, resetAxis := #resetAxis, openBrake := #openBrake, jogForward := #jogForward, jogBackward := #jogBackward, moveVelocity := #moveVelocity, stop := #stop, gearInVelocity := #gearInVelocity, torqueLimiting := #torqueLimiting, homing := #homing, posRelative := #posRelative, posAbsolute := #posAbsolute, posSuperimposed := #posSuperimposed, gearInRelatif := #gearInRelative, gearInAbsolute := #gearInAbsolute, camIn := #camIn, camInStandStill := #camInStandStill, phasing := #phasing, gearOutCamOut := #gearOutCamOut, actDeactLimitSwitches := #actDesactLimitSwitches, changeModulo := #changeModulo, homingToFixedStop := #homingToFixedStop, homingOnSensor := #homingOnSensor, resetMaxValues := #resetMaxValues, eStop := #eStop, StartEndLessMode := #startEndLessMode, camInChangeOnTheFly := #camInChangeOnTheFly, offset := #offset, haltSuperimposed := #haltSuperimposed, axisCommandStatusDWord => #statAxisCommandStatusDWord)
   END_RUNG
   // the same network as SCL:
   #instLaxisCtrlApcFr_GetCommandAxisStatusDWord(simulationOnoff := #simulationOnOff,   // "LAxisCtrlApcFr_GetCommandAxisStatusDWord"
                           stateSafetyActive := #stateSafetyActive,
                           stateS120InfeedInOperation := #stateS120InfeedInOperation,
                           enableAxis := #enableAxis,
                           resetAxis := #resetAxis,
                           openBrake := #openBrake,
                           jogForward := #jogForward,
                           jogBackward := #jogBackward,
                           moveVelocity := #moveVelocity,
                           stop := #stop,
                           gearInVelocity := #gearInVelocity,
                           torqueLimiting := #torqueLimiting,
                           homing := #homing,
                           posRelative := #posRelative,
                           posAbsolute := #posAbsolute,
                           posSuperimposed := #posSuperimposed,
                           gearInRelatif := #gearInRelative,
                           gearInAbsolute := #gearInAbsolute,
                           camIn := #camIn,
                           camInStandStill := #camInStandStill,
                           phasing := #phasing,
                           gearOutCamOut := #gearOutCamOut,
                           actDeactLimitSwitches := #actDesactLimitSwitches,
                           changeModulo := #changeModulo,
                           homingToFixedStop := #homingToFixedStop,
                           homingOnSensor := #homingOnSensor,
                           resetMaxValues := #resetMaxValues,
                           eStop := #eStop,
                           StartEndLessMode := #startEndLessMode,
                           camInChangeOnTheFly := #camInChangeOnTheFly,
                           offset := #offset,
                           haltSuperimposed := #haltSuperimposed,
                           axisCommandStatusDWord => #statAxisCommandStatusDWord);
END_REGION

REGION Network 24: (** OUTPUT AXIS STATE **)
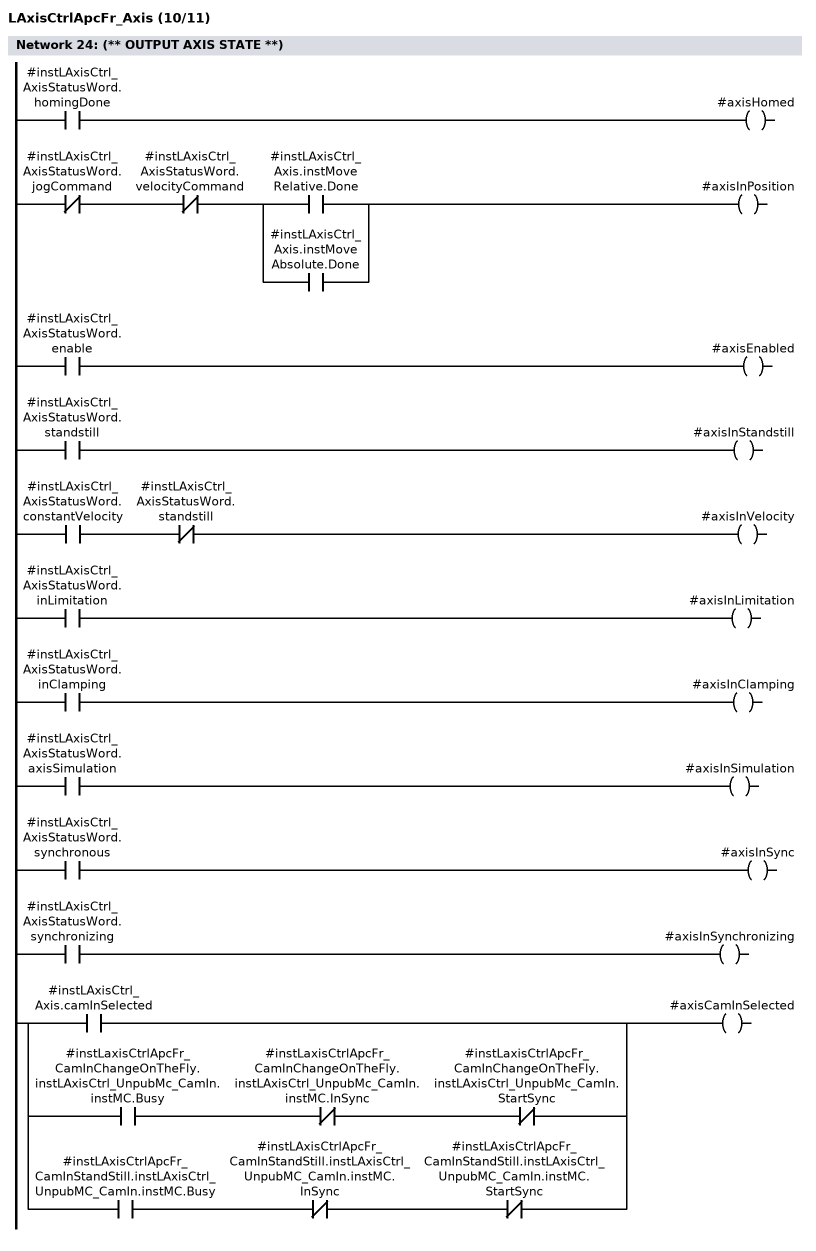
   RUNG wire#powerrail
      Contact( #instLAxisCtrl_AxisStatusWord.homingDone )
      Coil( #axisHomed )
   END_RUNG
   RUNG wire#powerrail
      I_Contact( #instLAxisCtrl_AxisStatusWord.jogCommand )
      I_Contact( #instLAxisCtrl_AxisStatusWord.velocityCommand )
      wire#w1
      Contact( #instLAxisCtrl_Axis.instMoveRelative.Done )
      wire#w2
      Coil( #axisInPosition )
   END_RUNG
   RUNG wire#w1
      Contact( #instLAxisCtrl_Axis.instMoveAbsolute.Done )
   END_RUNG wire#w2
   RUNG wire#powerrail
      Contact( #instLAxisCtrl_AxisStatusWord.enable )
      Coil( #axisEnabled )
   END_RUNG
   RUNG wire#powerrail
      Contact( #instLAxisCtrl_AxisStatusWord.standstill )
      Coil( #axisInStandstill )
   END_RUNG
   RUNG wire#powerrail
      Contact( #instLAxisCtrl_AxisStatusWord.constantVelocity )
      I_Contact( #instLAxisCtrl_AxisStatusWord.standstill )
      Coil( #axisInVelocity )
   END_RUNG
   RUNG wire#powerrail
      Contact( #instLAxisCtrl_AxisStatusWord.inLimitation )
      Coil( #axisInLimitation )
   END_RUNG
   RUNG wire#powerrail
      Contact( #instLAxisCtrl_AxisStatusWord.inClamping )
      Coil( #axisInClamping )
   END_RUNG
   RUNG wire#powerrail
      Contact( #instLAxisCtrl_AxisStatusWord.axisSimulation )
      Coil( #axisInSimulation )
   END_RUNG
   RUNG wire#powerrail
      Contact( #instLAxisCtrl_AxisStatusWord.synchronous )
      Coil( #axisInSync )
   END_RUNG
   RUNG wire#powerrail
      Contact( #instLAxisCtrl_AxisStatusWord.synchronizing )
      Coil( #axisInSynchronizing )
   END_RUNG
   RUNG wire#powerrail
      Contact( #instLAxisCtrl_Axis.camInSelected )
      wire#w3
      Coil( #axisCamInSelected )
   END_RUNG
   RUNG wire#powerrail
      Contact( #instLaxisCtrlApcFr_CamInChangeOnTheFly.instLAxisCtrl_UnpubMc_CamIn.instMC.Busy )
      I_Contact( #instLaxisCtrlApcFr_CamInChangeOnTheFly.instLAxisCtrl_UnpubMc_CamIn.instMC.InSync )
      I_Contact( #instLaxisCtrlApcFr_CamInChangeOnTheFly.instLAxisCtrl_UnpubMc_CamIn.StartSync )
   END_RUNG wire#w3
   RUNG wire#powerrail
      Contact( #instLAxisCtrlApcFr_CamInStandStill.instLAxisCtrl_UnpubMC_CamIn.instMC.Busy )
      I_Contact( #instLAxisCtrlApcFr_CamInStandStill.instLAxisCtrl_UnpubMC_CamIn.instMC.InSync )
      I_Contact( #instLAxisCtrlApcFr_CamInStandStill.instLAxisCtrl_UnpubMC_CamIn.instMC.StartSync )
   END_RUNG wire#w3
   // the same network as SCL:
   #axisHomed := #instLAxisCtrl_AxisStatusWord.homingDone;
   #axisInPosition := NOT #instLAxisCtrl_AxisStatusWord.jogCommand AND NOT #instLAxisCtrl_AxisStatusWord.velocityCommand AND (#instLAxisCtrl_Axis.instMoveRelative.Done OR #instLAxisCtrl_Axis.instMoveAbsolute.Done);
   #axisEnabled := #instLAxisCtrl_AxisStatusWord.enable;
   #axisInStandstill := #instLAxisCtrl_AxisStatusWord.standstill;
   #axisInVelocity := #instLAxisCtrl_AxisStatusWord.constantVelocity AND NOT #instLAxisCtrl_AxisStatusWord.standstill;
   #axisInLimitation := #instLAxisCtrl_AxisStatusWord.inLimitation;
   #axisInClamping := #instLAxisCtrl_AxisStatusWord.inClamping;
   #axisInSimulation := #instLAxisCtrl_AxisStatusWord.axisSimulation;
   #axisInSync := #instLAxisCtrl_AxisStatusWord.synchronous;
   #axisInSynchronizing := #instLAxisCtrl_AxisStatusWord.synchronizing;
   #axisCamInSelected := #instLAxisCtrl_Axis.camInSelected OR (#instLaxisCtrlApcFr_CamInChangeOnTheFly.instLAxisCtrl_UnpubMc_CamIn.instMC.Busy AND NOT #instLaxisCtrlApcFr_CamInChangeOnTheFly.instLAxisCtrl_UnpubMc_CamIn.instMC.InSync AND NOT #instLaxisCtrlApcFr_CamInChangeOnTheFly.instLAxisCtrl_UnpubMc_CamIn.StartSync) OR (#instLAxisCtrlApcFr_CamInStandStill.instLAxisCtrl_UnpubMC_CamIn.instMC.Busy AND NOT #instLAxisCtrlApcFr_CamInStandStill.instLAxisCtrl_UnpubMC_CamIn.instMC.InSync AND NOT #instLAxisCtrlApcFr_CamInStandStill.instLAxisCtrl_UnpubMC_CamIn.instMC.StartSync);
END_REGION

REGION Network 25 (SCL): (** OUTPUT CAM STATE **)
   #tempRefSyncAxis ?= #axis;

   IF #tempRefSyncAxis <> NULL THEN
       IF #tempRefSyncAxis^.StatusSynchronizedMotion.ActualCam = #cam1 AND #cam1 <> 0 THEN
           #camUsed := 1;
       ELSIF #tempRefSyncAxis^.StatusSynchronizedMotion.ActualCam = #cam2 AND #cam2 <> 0 THEN
           #camUsed := 2;
       ELSE
           #camUsed := 0;
       END_IF;
   END_IF;
END_REGION

REGION Network 26: (** DRIVE READY FOR OPERATION **)
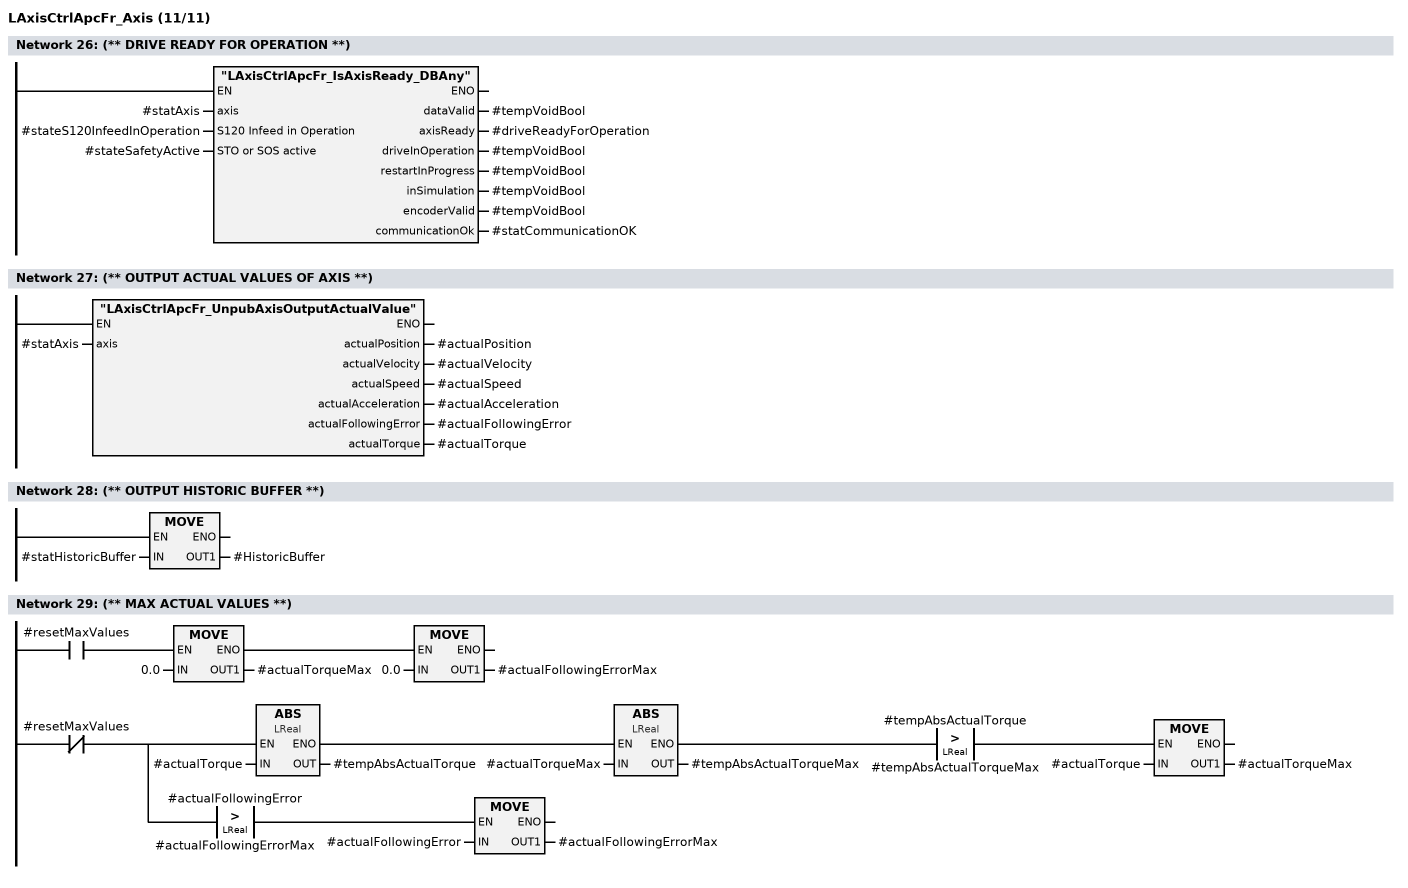
   RUNG wire#powerrail
      "LAxisCtrlApcFr_IsAxisReady_DBAny"(axis := #statAxis, "S120 Infeed in Operation" := #stateS120InfeedInOperation, "STO or SOS active" := #stateSafetyActive, dataValid => #tempVoidBool, axisReady => #driveReadyForOperation, driveInOperation => #tempVoidBool, restartInProgress => #tempVoidBool, inSimulation => #tempVoidBool, encoderValid => #tempVoidBool, communicationOk => #statCommunicationOK)
   END_RUNG
   // the same network as SCL:
   "LAxisCtrlApcFr_IsAxisReady_DBAny"(axis := #statAxis,
                           "S120 Infeed in Operation" := #stateS120InfeedInOperation,
                           "STO or SOS active" := #stateSafetyActive,
                           dataValid => #tempVoidBool,
                           axisReady => #driveReadyForOperation,
                           driveInOperation => #tempVoidBool,
                           restartInProgress => #tempVoidBool,
                           inSimulation => #tempVoidBool,
                           encoderValid => #tempVoidBool,
                           communicationOk => #statCommunicationOK);
END_REGION

REGION Network 27: (** OUTPUT ACTUAL VALUES OF AXIS **)
   RUNG wire#powerrail
      "LAxisCtrlApcFr_UnpubAxisOutputActualValue"(axis := #statAxis, actualPosition => #actualPosition, actualVelocity => #actualVelocity, actualSpeed => #actualSpeed, actualAcceleration => #actualAcceleration, actualFollowingError => #actualFollowingError, actualTorque => #actualTorque)
   END_RUNG
   // the same network as SCL:
   "LAxisCtrlApcFr_UnpubAxisOutputActualValue"(axis := #statAxis,
                           actualPosition => #actualPosition,
                           actualVelocity => #actualVelocity,
                           actualSpeed => #actualSpeed,
                           actualAcceleration => #actualAcceleration,
                           actualFollowingError => #actualFollowingError,
                           actualTorque => #actualTorque);
END_REGION

REGION Network 28: (** OUTPUT HISTORIC BUFFER **)
   RUNG wire#powerrail
      Move(in := #statHistoricBuffer, out1 => #HistoricBuffer)
   END_RUNG
   // the same network as SCL:
   #HistoricBuffer := #statHistoricBuffer;
END_REGION

REGION Network 29: (** MAX ACTUAL VALUES **)
   RUNG wire#powerrail
      Contact( #resetMaxValues )
      Move(in := 0.0, out1 => #actualTorqueMax)
      Move(in := 0.0, out1 => #actualFollowingErrorMax)
   END_RUNG
   RUNG wire#powerrail
      I_Contact( #resetMaxValues )
      wire#w1
      { S7_Templates := "SrcType := LReal" } Abs(in := #actualTorque, out => #tempAbsActualTorque)
      { S7_Templates := "SrcType := LReal" } Abs(in := #actualTorqueMax, out => #tempAbsActualTorqueMax)
      { S7_Templates := "SrcType := LReal" } GT_Contact(in1 := #tempAbsActualTorque, in2 := #tempAbsActualTorqueMax)
      Move(in := #actualTorque, out1 => #actualTorqueMax)
   END_RUNG
   RUNG wire#w1
      { S7_Templates := "SrcType := LReal" } GT_Contact(in1 := #actualFollowingError, in2 := #actualFollowingErrorMax)
      Move(in := #actualFollowingError, out1 => #actualFollowingErrorMax)
   END_RUNG
   // the same network as SCL:
   IF #resetMaxValues THEN
       #actualTorqueMax := 0.0;
       #actualFollowingErrorMax := 0.0;
   END_IF;
   IF NOT #resetMaxValues THEN
       #tempAbsActualTorque := ABS(#actualTorque);
       #tempAbsActualTorqueMax := ABS(#actualTorqueMax);
   END_IF;
   IF NOT #resetMaxValues AND (#tempAbsActualTorque > #tempAbsActualTorqueMax) THEN
       #actualTorqueMax := #actualTorque;
   END_IF;
   IF NOT #resetMaxValues AND (#actualFollowingError > #actualFollowingErrorMax) THEN
       #actualFollowingErrorMax := #actualFollowingError;
   END_IF;
END_REGION

REGION Network 30 (SCL): (** ERROR **)
   //----------------------------------------------------------------------------------------------
   IF NOT #statFirstError THEN

       // ERROR TO AXIS
       IF #instLAxisCtrl_AxisStatusWord.error THEN
           REGION ----- Error GetAxisStatusWord -----
               // Diagnostic in string
               #status := 'ERR_TO_AXIS';
               #errorMC := 'No error MC instruction';
               #errorID := "LAxisCtrlApcFr_Word2String_TO.ErrorDetailNumber"(errorDetailNumber := "LAxisCtrlApcFr_UnpubAxisErrorDetailNumber"(#statAxis), language := #dataAxisConfig.textLanguage);
               // Diagnostic in word
               #statDiagnostic.status := "ERR_LAXISCTRLAPCFR_TO_AXIS";
               #statDiagnostic.errorMC := "STATUS_FINISHED_NOERROR";
               #statDiagnostic.errorID := UDINT_TO_WORD("LAxisCtrlApcFr_UnpubAxisErrorDetailNumber"(#statAxis));

               #error := TRUE;
               #statFirstError := TRUE;
           END_REGION

       // ERROR LAXISCTRL STANDARD
       ELSIF #statErrorLAxisCtrlStd THEN
           REGION ----- ErrorLAxisCtrlStd -----
               // Diagnostic in string
               #status := "LAxisCtrlApcFr_Word2String_Status"(wordStatus := "ERR_LAXISCTRLAPCFR_LAXISCTRL");
               #errorMC := "LAxisCtrlApcFr_Word2String_LaxisCtrl.Status"(wordStatus := #instLAxisCtrl_Axis.diagnostics.status, language := #dataAxisConfig.textLanguage);
               #errorID := "LAxisCtrlApcFr_Word2String_ErrorID"(wordErrorID := #instLAxisCtrl_Axis.diagnostics.subfunctionStatus, language := #dataAxisConfig.textLanguage);
               // Diagnostic in word
               #statDiagnostic.status := "ERR_LAXISCTRLAPCFR_LAXISCTRL";
               #statDiagnostic.errorMC := #instLAxisCtrl_Axis.diagnostics.status;
               #statDiagnostic.errorID := #instLAxisCtrl_Axis.diagnostics.subfunctionStatus;

               #error := TRUE;
               #statFirstError := TRUE;
           END_REGION

       // ERROR DRIVE AND ENCODER COMMUNICATION
       ELSIF NOT #statCommunicationOK AND #homing THEN
           REGION ----- ErrorLAxisCtrlStd -----
               // Diagnostic in string
               #status := "LAxisCtrlApcFr_Word2String_Status"(wordStatus := "ERR_LAXISCTRLAPCFR_HOMING_WITH_DRIVE_AND_ENCODER_COMMUNICATION_NOK");
               #errorMC := 'No errorMC';
               #errorID := "LAxisCtrlApcFr_Word2String_Status"(wordStatus := "ERR_LAXISCTRLAPCFR_NO_DRIVE_AND_ENCODER_COMMUNICATION");
               // Diagnostic in word
               #statDiagnostic.status := "ERR_LAXISCTRLAPCFR_HOMING_WITH_DRIVE_AND_ENCODER_COMMUNICATION_NOK";
               #statDiagnostic.errorMC := "STATUS_FINISHED_NOERROR";
               #statDiagnostic.errorID := "ERR_LAXISCTRLAPCFR_NO_DRIVE_AND_ENCODER_COMMUNICATION";

               #error := TRUE;
               #statFirstError := TRUE;
           END_REGION

       // ERROR DRIVE IN OPERATION
       ELSIF NOT #driveReadyForOperation AND #enableAxis AND NOT #instLAxisCtrl_AxisStatusWord.axisSimulation THEN
           REGION ----- Error enableAxis without driveReadyForOperation -----
               // Diagnostic in string
               #status := "LAxisCtrlApcFr_Word2String_Status"(wordStatus := "ERR_LAXISCTRLAPCFR_POWERON_WITH_DRIVE_NO_READY");
               #errorMC := 'No errorMC';
               IF NOT #statCommunicationOK THEN //"LAxisCtrlApcFr_UnpubAxisStatusDriveCommunicationOK"(#statAxis) THEN
                   #errorID := "LAxisCtrlApcFr_Word2String_Status"(wordStatus := "ERR_LAXISCTRLAPCFR_NO_DRIVE_AND_ENCODER_COMMUNICATION");
                   #statDiagnostic.errorID := "ERR_LAXISCTRLAPCFR_NO_DRIVE_AND_ENCODER_COMMUNICATION";
               ELSIF #stateSafetyActive THEN
                   #errorID := "LAxisCtrlApcFr_Word2String_Status"(wordStatus := "ERR_LAXISCTRLAPCFR_SAFETY_ACTIVATED");
                   #statDiagnostic.errorID := "ERR_LAXISCTRLAPCFR_SAFETY_ACTIVATED";
               ELSIF NOT #stateS120InfeedInOperation THEN
                   #errorID := "LAxisCtrlApcFr_Word2String_Status"(wordStatus := "ERR_LAXISCTRLAPCFR_NOT_INFEED_IN_OPERATION");
                   #statDiagnostic.errorID := "ERR_LAXISCTRLAPCFR_NOT_INFEED_IN_OPERATION";
               END_IF;
               // Diagnostic in Word
               #statDiagnostic.status := "ERR_LAXISCTRLAPCFR_POWERON_WITH_DRIVE_NO_READY";
               #statDiagnostic.errorMC := "STATUS_FINISHED_NOERROR";

               #error := TRUE;
               #statFirstError := TRUE;
           END_REGION

       // ERROR ESTOP
       ELSIF #statErrorEStop THEN
           REGION ----- Error MC_Stop -----
               // Diagnostic in string
               #status := "LAxisCtrlApcFr_Word2String_Status"(wordStatus := "ERR_LAXISCTRLAPCFR_ESTOP");
               #errorMC := "LAxisCtrlApcFr_Word2String_Status"(wordStatus := "ERR_LAXISCTRLAPCFR_ESTOP_IN_ERROR");
               #errorID := "LAxisCtrlApcFr_Word2String_ErrorID"(wordErrorID := #instLAxisCtrlApcFr_UnpubAxis_eSTOP.errorId, language := #dataAxisConfig.textLanguage);
               // Diagnostic in word
               #statDiagnostic.status := "ERR_LAXISCTRLAPCFR_ESTOP";
               #statDiagnostic.errorMC := "ERR_LAXISCTRLAPCFR_ESTOP_IN_ERROR";
               #statDiagnostic.errorID := #instLAxisCtrlApcFr_UnpubAxis_eSTOP.errorId;

               #error := TRUE;
               #statFirstError := TRUE;
           END_REGION

       // ERROR HOMING TO FIXED STOP
       ELSIF #statErrorHomingToFixedStop THEN
           REGION ----- ErrorHomingTorque -----
               // Diagnostic in string
               #status := "LAxisCtrlApcFr_Word2String_Status"(wordStatus := "ERR_LAXISCTRLAPCFR_HOMING_TO_FIXED_STOP");
               #errorMC := "LAxisCtrlApcFr_Word2String_Status"(wordStatus:=#instLAxisCtrlApcFr_HomingToFixedStop.status);
               #errorID := "LAxisCtrlApcFr_Word2String_ErrorID"(wordErrorID:=#instLAxisCtrlApcFr_HomingToFixedStop.subStatus, language:=#dataAxisConfig.textLanguage);
               // Diagnostic in word
               #statDiagnostic.status := "ERR_LAXISCTRLAPCFR_HOMING_TO_FIXED_STOP";
               #statDiagnostic.errorMC := #instLAxisCtrlApcFr_HomingToFixedStop.status;
               #statDiagnostic.errorID := #instLAxisCtrlApcFr_HomingToFixedStop.subStatus;

               #error := TRUE;
               #statFirstError := TRUE;
           END_REGION

       // ERROR HOMING ON SENSOR
       ELSIF #statErrorHomingOnSensor THEN
           REGION ----- ErrorHomingOnSensor -----
               // Diagnostic in string
               #status := "LAxisCtrlApcFr_Word2String_Status"(wordStatus := "ERR_LAXISCTRLAPCFR_HOMING_ON_SENSOR");
               #errorMC := "LAxisCtrlApcFr_Word2String_Status"(wordStatus := #instAxisCtrlAapcFr_HomingOnSensor.status);
               #errorID := "LAxisCtrlApcFr_Word2String_ErrorID"(wordErrorID := #instAxisCtrlAapcFr_HomingOnSensor.subStatus, language := #dataAxisConfig.textLanguage);
               // Diagnostic in word
               #statDiagnostic.status := "ERR_LAXISCTRLAPCFR_HOMING_ON_SENSOR";
               #statDiagnostic.errorMC := #instAxisCtrlAapcFr_HomingOnSensor.status;
               #statDiagnostic.errorID := #instAxisCtrlAapcFr_HomingOnSensor.subStatus;

               #error := TRUE;
               #statFirstError := TRUE;
           END_REGION

       //ERROR ACT DESACT LIMIT SWITCHES
       ELSIF #statErrorActDesactLimitSwitches THEN
           REGION ----- ErrorActLimitSwitches -----
               // Diagnostic in string
               #status := "LAxisCtrlApcFr_Word2String_Status"(wordStatus := "ERR_LAXISCTRLAPCFR_ACT_LIMIT_SWITCHES");
               #errorMC := "LAxisCtrlApcFr_Word2String_Status"(wordStatus := #instLAxisCtrlApcFr_ActDeactLimitSwitches.status);
               #errorID := "LAxisCtrlApcFr_Word2String_ErrorID"(wordErrorID := #instLAxisCtrlApcFr_ActDeactLimitSwitches.subStatus, language := #dataAxisConfig.textLanguage);
               // Diagnostic in word
               #statDiagnostic.status := "ERR_LAXISCTRLAPCFR_ACT_LIMIT_SWITCHES";
               #statDiagnostic.errorMC := #instLAxisCtrlApcFr_ActDeactLimitSwitches.status;
               #statDiagnostic.errorID := #instLAxisCtrlApcFr_ActDeactLimitSwitches.subStatus;

               #error := TRUE;
               #statFirstError := TRUE;
           END_REGION

       // ERROR CHANGE MODULO
       ELSIF #statErrorChangeModuloAxis THEN
           REGION ----- ErrorChangeModuloAxis -----
               // Diagnostic in string
               #status := "LAxisCtrlApcFr_Word2String_Status"(wordStatus := "ERR_LAXISCTRLAPCFR_CHANGE_MODULO_AXIS");
               #errorMC := "LAxisCtrlApcFr_Word2String_Status"(wordStatus := #instLAxisCtrlApcFr_ChangeModulo.status);
               #errorID := "LAxisCtrlApcFr_Word2String_ErrorID"(wordErrorID := #instLAxisCtrlApcFr_ChangeModulo.subStatus, language := #dataAxisConfig.textLanguage);
               // Diagnostic in word
               #statDiagnostic.status := "ERR_LAXISCTRLAPCFR_CHANGE_MODULO_AXIS";
               #statDiagnostic.errorMC := #instLAxisCtrlApcFr_ChangeModulo.status;
               #statDiagnostic.errorID := #instLAxisCtrlApcFr_ChangeModulo.subStatus;

               #error := TRUE;
               #statFirstError := TRUE;
           END_REGION

       // ERROR ENDLESS MODE
       ELSIF #statErrorEndLessMode THEN
           REGION ----- ErrorStartEndLessMode -----
               // Diagnostic in string
               #status := "LAxisCtrlApcFr_Word2String_Status"(wordStatus := "ERR_LAXISCTRLAPCFR_ENDLESS_MODE");
               #errorMC := "LAxisCtrlApcFr_Word2String_Status"(wordStatus := #instLAxisCtrlApcFr_EndLessMode.status);
               #errorID := "LAxisCtrlApcFr_Word2String_ErrorID"(wordErrorID := #instLAxisCtrlApcFr_EndLessMode.subStatus, language := #dataAxisConfig.textLanguage);
               // Diagnostic in word
               #statDiagnostic.status := "ERR_LAXISCTRLAPCFR_ENDLESS_MODE";
               #statDiagnostic.errorMC := #instLAxisCtrlApcFr_EndLessMode.status;
               #statDiagnostic.errorID := #instLAxisCtrlApcFr_EndLessMode.subStatus;

               #error := TRUE;
               #statFirstError := TRUE;
           END_REGION

       // ERROR SIMULATION ON
       ELSIF #statErrorSimulationOnOff THEN
           REGION ----- ErrorSimulationOn -----
               // Diagnostic in string
               #status := "LAxisCtrlApcFr_Word2String_Status"(wordStatus := "ERR_LAXISCTRLAPCFR_SIMULATION_ON");
               #errorMC := "LAxisCtrlApcFr_Word2String_Status"(wordStatus := #instLAxisCtrlApcFR_SimulationOnOff.status);
               #errorID := "LAxisCtrlApcFr_Word2String_ErrorID"(wordErrorID := #instLAxisCtrlApcFR_SimulationOnOff.subStatus, language := #dataAxisConfig.textLanguage);
               // Diagnostic in word
               #statDiagnostic.status := "ERR_LAXISCTRLAPCFR_SIMULATION_ON";
               #statDiagnostic.errorMC := #instLAxisCtrlApcFR_SimulationOnOff.status;
               #statDiagnostic.errorID := #instLAxisCtrlApcFR_SimulationOnOff.subStatus;

               #error := TRUE;
               #statFirstError := TRUE;
           END_REGION

       //ERROR GEARINPOS
       ELSIF #statErrorGearInPos THEN
           REGION ----- ErrorGearInPos -----
               // Diagnostic in string
               #status := "LAxisCtrlApcFr_Word2String_Status"(wordStatus := "ERR_LAXISCTRLAPCFR_GEARINPOS");
               #errorMC := "LAxisCtrlApcFr_Word2String_Status"(wordStatus := #InstLAxisCtrlApcFr_McGearInPos_Axis.status);
               #errorID := "LAxisCtrlApcFr_Word2String_ErrorID"(wordErrorID := #InstLAxisCtrlApcFr_McGearInPos_Axis.subStatus, language := #dataAxisConfig.textLanguage);
               // Diagnostic in word
               #statDiagnostic.status := "ERR_LAXISCTRLAPCFR_GEARINPOS";
               #statDiagnostic.errorMC := #InstLAxisCtrlApcFr_McGearInPos_Axis.status;
               #statDiagnostic.errorID := #InstLAxisCtrlApcFr_McGearInPos_Axis.subStatus;

               #error := TRUE;
               #statFirstError := TRUE;
           END_REGION


